  MoveL 760 to (-510.72, -291.87, 844) mm, rotated rx 180 ry 0 rz -90 deg; joints [21.183, -72.621, -92.099, -15.28, 68.817, -90]
  MoveL 761 to (-508.3, -277.31, 840) mm, rotated rx 180 ry 0 rz -90 deg; joints [21.364, -72.698, -94.24, -13.063, 68.636, -90]
  MoveL 762 to (-516.77, -268.54, 854) mm, rotated rx 180 ry 0 rz -90 deg; joints [20.699, -70.474, -96.997, -12.53, 69.301, -90]
  MoveL 763 to (-516.77, -255.15, 854) mm, rotated rx 180 ry 0 rz -90 deg; joints [20.699, -70.107, -99.223, -10.67, 69.301, -90]
  MoveL 764 to (-526.45, -246.29, 870) mm, rotated rx 180 ry 0 rz -90 deg; joints [19.827, -67.632, -102.031, -10.337, 70.173, -90]
  MoveL 765 to (-521.61, -230.51, 862) mm, rotated rx 180 ry 0 rz -90 deg; joints [20.28, -68.427, -103.896, -7.678, 69.72, -90]
  MoveL 766 to (-519.19, -215.98, 858) mm, rotated rx 180 ry 0 rz -90 deg; joints [20.493, -68.776, -105.82, -5.404, 69.507, -90]
  MoveL 767 to (-527.05, -205.6, 871) mm, rotated rx 180 ry 0 rz -90 deg; joints [19.768, -66.744, -108.538, -4.718, 70.232, -90]
  MoveL 768 to (-525.24, -191.28, 868) mm, rotated rx 180 ry 0 rz -90 deg; joints [19.944, -67.058, -110.452, -2.489, 70.056, -90]
  MoveL 769 to (-524.63, -177.46, 867) mm, rotated rx 180 ry 0 rz -90 deg; joints [20.001, -67.158, -112.413, -0.43, 69.999, -90]
  MoveL 770 to (-527.66, -164.81, 872) mm, rotated rx 180 ry 0 rz -90 deg; joints [19.709, -66.408, -114.69, 1.097, 70.291, -90]
  MoveL 771 to (-528.26, -151.31, 873) mm, rotated rx 180 ry 0 rz -90 deg; joints [19.649, -66.326, -116.708, 3.035, 70.351, -90]
  MoveL 772 to (-527.66, -137.46, 872) mm, rotated rx 180 ry 0 rz -90 deg; joints [19.709, -66.634, -118.561, 5.195, 70.291, -90]
  MoveL 773 to (-533.71, -125.21, 882) mm, rotated rx 180 ry 0 rz -90 deg; joints [19.079, -65.242, -121.134, 6.376, 70.921, -90]
  MoveL 774 to (-526.45, -109.86, 870) mm, rotated rx 180 ry 0 rz -90 deg; joints [19.827, -67.51, -122.122, 9.633, 70.173, -90]
  MoveL 775 to (-527.66, -96.44, 872) mm, rotated rx 180 ry 0 rz -90 deg; joints [19.709, -67.583, -124.075, 11.657, 70.291, -90]
  MoveL 776 to (-521.61, -81.82, 862) mm, rotated rx 180 ry 0 rz -90 deg; joints [20.28, -69.783, -124.958, 14.74, 69.72, -90]
  MoveL 777 to (-528.26, -69.17, 873) mm, rotated rx 180 ry 0 rz -90 deg; joints [19.649, -68.506, -127.639, 16.145, 70.351, -90]
  MoveL 778 to (-520.4, -54.65, 860) mm, rotated rx 180 ry 0 rz -90 deg; joints [20.388, -71.46, -128.062, 19.522, 69.612, -90]
  MoveL 779 to (-517.98, -40.98, 856) mm, rotated rx 180 ry 0 rz -90 deg; joints [20.597, -72.977, -129.219, 22.196, 69.403, -90]
  MoveL 780 to (-511.93, -27.23, 846) mm, rotated rx 180 ry 0 rz -90 deg; joints [21.089, -75.629, -129.608, 25.237, 68.911, -90]
  MoveL 781 to (-506.48, -13.82, 837) mm, rotated rx 180 ry 0 rz -90 deg; joints [21.496, -78.189, -129.943, 28.132, 68.504, -90]
  MoveL 782 to (-507.69, -0.69, 839) mm, rotated rx 180 ry 0 rz -90 deg; joints [21.409, -79.002, -131.528, 30.53, 68.591, -90]
  MoveL 783 to (-504.66, 12.39, 834) mm, rotated rx 180 ry 0 rz -90 deg; joints [21.625, -81.074, -132.163, 33.237, 68.375, -90]
  MoveL 784 to (-503.45, 25.41, 832) mm, rotated rx 180 ry 0 rz -90 deg; joints [21.709, -82.751, -133.104, 35.855, 68.291, -90]
  MoveL 785 to (-498.61, 38.08, 824) mm, rotated rx 180 ry 0 rz -90 deg; joints [22.032, -85.434, -133.121, 38.554, 67.969, -90]
  MoveL 786 to (-496.19, 50.76, 820) mm, rotated rx 180 ry 0 rz -90 deg; joints [22.185, -87.555, -133.593, 41.148, 67.815, -90]
  MoveL 787 to (-491.35, 63, 812) mm, rotated rx 180 ry 0 rz -90 deg; joints [22.478, -90.28, -133.363, 43.643, 67.522, -90]
  MoveL 788 to (-489.54, 75.45, 809) mm, rotated rx 180 ry 0 rz -90 deg; joints [22.583, -92.346, -133.791, 46.137, 67.418, -90]
  MoveL 789 to (-481.67, 86.72, 796) mm, rotated rx 180 ry 0 rz -90 deg; joints [23.011, -95.661, -132.528, 48.189, 66.989, -90]
  MoveL 790 to (-479.85, 98.83, 793) mm, rotated rx 180 ry 0 rz -90 deg; joints [23.104, -97.738, -132.762, 50.5, 66.896, -90]
  MoveL 791 to (-478.04, 110.84, 790) mm, rotated rx 180 ry 0 rz -90 deg; joints [23.195, -99.846, -132.917, 52.764, 66.805, -90]
  MoveL 792 to (-476.22, 122.76, 787) mm, rotated rx 180 ry 0 rz -90 deg; joints [23.284, -101.979, -132.995, 54.974, 66.717, -90]
  MoveL 793 to (-499.84, -492.72, 848) mm, rotated rx 180 ry 0 rz -90 deg; joints [23.844, -86.996, -46.335, -46.669, 66.156, -90]
  MoveL 794 to (-495.71, -475.46, 841) mm, rotated rx 180 ry 0 rz -90 deg; joints [24.056, -85.782, -50.992, -43.226, 65.944, -90]
  MoveL 795 to (-492.18, -458.98, 835) mm, rotated rx 180 ry 0 rz -90 deg; joints [24.228, -84.764, -55.111, -40.125, 65.772, -90]
  MoveL 796 to (-498.07, -451.22, 845) mm, rotated rx 180 ry 0 rz -90 deg; joints [23.937, -82.603, -58.407, -38.99, 66.063, -90]
  MoveL 797 to (-496.89, -436.94, 843) mm, rotated rx 180 ry 0 rz -90 deg; joints [23.997, -81.512, -61.93, -36.557, 66.003, -90]
  MoveL 798 to (-491.59, -419.19, 834) mm, rotated rx 180 ry 0 rz -90 deg; joints [24.256, -81.2, -65.344, -33.456, 65.744, -90]
  MoveL 799 to (-494.53, -408.55, 839) mm, rotated rx 180 ry 0 rz -90 deg; joints [24.114, -79.678, -68.387, -31.935, 65.886, -90]
  MoveL 800 to (-490.41, -392.09, 832) mm, rotated rx 180 ry 0 rz -90 deg; joints [24.311, -79.429, -71.37, -29.201, 65.69, -90]
  MoveL 801 to (-491, -379.5, 833) mm, rotated rx 180 ry 0 rz -90 deg; joints [24.283, -78.45, -74.205, -27.345, 65.717, -90]
  MoveL 802 to (-492.18, -367.32, 835) mm, rotated rx 180 ry 0 rz -90 deg; joints [24.228, -77.42, -76.962, -25.618, 65.772, -90]
  MoveL 803 to (-491.59, -353.8, 834) mm, rotated rx 180 ry 0 rz -90 deg; joints [24.256, -76.782, -79.601, -23.616, 65.744, -90]
  MoveL 804 to (-494.53, -342.77, 839) mm, rotated rx 180 ry 0 rz -90 deg; joints [24.114, -75.504, -82.269, -22.227, 65.886, -90]
  MoveL 805 to (-492.76, -328.43, 836) mm, rotated rx 180 ry 0 rz -90 deg; joints [24.2, -75.22, -84.714, -20.066, 65.8, -90]
  MoveL 806 to (-498.66, -319.09, 846) mm, rotated rx 180 ry 0 rz -90 deg; joints [23.906, -73.399, -87.416, -19.185, 66.094, -90]
  MoveL 807 to (-497.48, -305.1, 844) mm, rotated rx 180 ry 0 rz -90 deg; joints [23.967, -73.091, -89.772, -17.136, 66.033, -90]
  MoveL 808 to (-499.84, -293.25, 848) mm, rotated rx 180 ry 0 rz -90 deg; joints [23.844, -72.074, -92.25, -15.676, 66.156, -90]
  MoveL 809 to (-496.89, -278.3, 843) mm, rotated rx 180 ry 0 rz -90 deg; joints [23.997, -72.283, -94.367, -13.35, 66.003, -90]
  MoveL 810 to (-497.48, -265.4, 844) mm, rotated rx 180 ry 0 rz -90 deg; joints [23.967, -71.761, -96.64, -11.599, 66.033, -90]
  MoveL 811 to (-506.32, -256.64, 859) mm, rotated rx 180 ry 0 rz -90 deg; joints [23.482, -69.341, -99.474, -11.185, 66.518, -90]
  MoveL 812 to (-511.63, -245.72, 868) mm, rotated rx 180 ry 0 rz -90 deg; joints [23.156, -67.749, -102.047, -10.204, 66.844, -90]
  MoveL 813 to (-510.45, -231.58, 866) mm, rotated rx 180 ry 0 rz -90 deg; joints [23.231, -67.732, -104.149, -8.119, 66.769, -90]
  MoveL 814 to (-513.98, -219.51, 872) mm, rotated rx 180 ry 0 rz -90 deg; joints [23.002, -66.616, -106.57, -6.815, 66.998, -90]
  MoveL 815 to (-513.98, -205.83, 872) mm, rotated rx 180 ry 0 rz -90 deg; joints [23.002, -66.418, -108.688, -4.893, 66.998, -90]
  MoveL 816 to (-509.27, -190.39, 864) mm, rotated rx 180 ry 0 rz -90 deg; joints [23.304, -67.515, -110.316, -2.169, 66.696, -90]
  MoveL 817 to (-512.81, -178.07, 870) mm, rotated rx 180 ry 0 rz -90 deg; joints [23.08, -66.53, -112.683, -0.786, 66.92, -90]
  MoveL 818 to (-512.81, -164.43, 870) mm, rotated rx 180 ry 0 rz -90 deg; joints [23.08, -66.538, -114.671, 1.209, 66.92, -90]
  MoveL 819 to (-510.45, -150.1, 866) mm, rotated rx 180 ry 0 rz -90 deg; joints [23.231, -67.272, -116.344, 3.616, 66.769, -90]
  MoveL 820 to (-515.75, -137.93, 875) mm, rotated rx 180 ry 0 rz -90 deg; joints [22.882, -65.937, -118.884, 4.821, 67.118, -90]
  MoveL 821 to (-516.34, -124.35, 876) mm, rotated rx 180 ry 0 rz -90 deg; joints [22.841, -65.986, -120.85, 6.836, 67.159, -90]
  MoveL 822 to (-519.29, -111.25, 881) mm, rotated rx 180 ry 0 rz -90 deg; joints [22.631, -65.421, -123.091, 8.512, 67.369, -90]
  MoveL 823 to (-513.98, -96.44, 872) mm, rotated rx 180 ry 0 rz -90 deg; joints [23.002, -67.378, -124.193, 11.57, 66.998, -90]
  MoveL 824 to (-510.45, -82.2, 866) mm, rotated rx 180 ry 0 rz -90 deg; joints [23.231, -68.937, -125.412, 14.35, 66.769, -90]
  MoveL 825 to (-512.22, -68.85, 869) mm, rotated rx 180 ry 0 rz -90 deg; joints [23.118, -69.007, -127.391, 16.398, 66.882, -90]
  MoveL 826 to (-509.27, -54.91, 864) mm, rotated rx 180 ry 0 rz -90 deg; joints [23.304, -70.615, -128.553, 19.168, 66.696, -90]
  MoveL 827 to (-503.37, -40.88, 854) mm, rotated rx 180 ry 0 rz -90 deg; joints [23.651, -73.232, -129.066, 22.298, 66.349, -90]
  MoveL 828 to (-498.07, -27.2, 845) mm, rotated rx 180 ry 0 rz -90 deg; joints [23.937, -75.76, -129.521, 25.281, 66.063, -90]
  MoveL 829 to (-495.12, -13.87, 840) mm, rotated rx 180 ry 0 rz -90 deg; joints [24.086, -77.673, -130.319, 27.992, 65.914, -90]
  MoveL 830 to (-491.59, -0.69, 834) mm, rotated rx 180 ry 0 rz -90 deg; joints [24.256, -79.841, -130.884, 30.725, 65.744, -90]
  MoveL 831 to (-492.76, 12.42, 836) mm, rotated rx 180 ry 0 rz -90 deg; joints [24.2, -80.756, -132.421, 33.177, 65.8, -90]
  MoveL 832 to (-491.59, 25.47, 834) mm, rotated rx 180 ry 0 rz -90 deg; joints [24.256, -82.45, -133.364, 35.814, 65.744, -90]
  MoveL 833 to (-484.51, 37.99, 822) mm, rotated rx 180 ry 0 rz -90 deg; joints [24.571, -85.795, -132.78, 38.575, 65.429, -90]
  MoveL 834 to (-479.8, 50.39, 814) mm, rotated rx 180 ry 0 rz -90 deg; joints [24.765, -88.502, -132.621, 41.123, 65.235, -90]
  MoveL 835 to (-478.62, 63, 812) mm, rotated rx 180 ry 0 rz -90 deg; joints [24.811, -90.369, -133.273, 43.642, 65.189, -90]
  MoveL 836 to (-476.26, 75.36, 808) mm, rotated rx 180 ry 0 rz -90 deg; joints [24.902, -92.572, -133.53, 46.102, 65.098, -90]
  MoveL 837 to (-468.6, 86.61, 795) mm, rotated rx 180 ry 0 rz -90 deg; joints [25.178, -95.905, -132.221, 48.125, 64.822, -90]
  MoveL 838 to (-466.83, 98.7, 792) mm, rotated rx 180 ry 0 rz -90 deg; joints [25.239, -97.975, -132.441, 50.416, 64.761, -90]
  MoveL 839 to (-466.83, 111.12, 792) mm, rotated rx 180 ry 0 rz -90 deg; joints [25.239, -99.763, -133.094, 52.857, 64.761, -90]
  MoveL 840 to (-468.01, 123.86, 794) mm, rotated rx 180 ry 0 rz -90 deg; joints [25.199, -101.44, -134.021, 55.461, 64.801, -90]
  MoveL 841 to (-483.67, -489.81, 843) mm, rotated rx 180 ry 0 rz -90 deg; joints [26.705, -87.373, -46.601, -46.025, 63.295, -90]
  MoveL 842 to (-485.39, -478.29, 846) mm, rotated rx 180 ry 0 rz -90 deg; joints [26.662, -85.483, -50.688, -43.829, 63.338, -90]
  MoveL 843 to (-483.67, -463.37, 843) mm, rotated rx 180 ry 0 rz -90 deg; joints [26.705, -84.199, -54.753, -41.047, 63.295, -90]
  MoveL 844 to (-480.8, -447.49, 838) mm, rotated rx 180 ry 0 rz -90 deg; joints [26.775, -83.263, -58.557, -38.179, 63.225, -90]
  MoveL 845 to (-483.1, -436.42, 842) mm, rotated rx 180 ry 0 rz -90 deg; joints [26.72, -81.666, -61.901, -36.433, 63.28, -90]
  MoveL 846 to (-481.95, -422.21, 840) mm, rotated rx 180 ry 0 rz -90 deg; joints [26.748, -80.707, -65.206, -34.087, 63.252, -90]
  MoveL 847 to (-480.23, -407.58, 837) mm, rotated rx 180 ry 0 rz -90 deg; joints [26.789, -79.957, -68.338, -31.705, 63.211, -90]
  MoveL 848 to (-477.36, -392.09, 832) mm, rotated rx 180 ry 0 rz -90 deg; joints [26.855, -79.528, -71.294, -29.179, 63.145, -90]
  MoveL 849 to (-478.51, -379.96, 834) mm, rotated rx 180 ry 0 rz -90 deg; joints [26.829, -78.435, -74.142, -27.423, 63.171, -90]
  MoveL 850 to (-478.51, -366.88, 834) mm, rotated rx 180 ry 0 rz -90 deg; joints [26.829, -77.624, -76.882, -25.494, 63.171, -90]
  MoveL 851 to (-482.52, -356.77, 841) mm, rotated rx 180 ry 0 rz -90 deg; joints [26.734, -76.054, -79.653, -24.293, 63.266, -90]
  MoveL 852 to (-480.8, -342.36, 838) mm, rotated rx 180 ry 0 rz -90 deg; joints [26.775, -75.702, -82.193, -22.105, 63.225, -90]
  MoveL 853 to (-484.25, -331.57, 844) mm, rotated rx 180 ry 0 rz -90 deg; joints [26.691, -74.315, -84.854, -20.831, 63.309, -90]
  MoveL 854 to (-483.67, -317.96, 843) mm, rotated rx 180 ry 0 rz -90 deg; joints [26.705, -73.833, -87.297, -18.87, 63.295, -90]
  MoveL 855 to (-485.97, -306.19, 847) mm, rotated rx 180 ry 0 rz -90 deg; joints [26.647, -72.763, -89.826, -17.411, 63.353, -90]
  MoveL 856 to (-486.54, -293.25, 848) mm, rotated rx 180 ry 0 rz -90 deg; joints [26.632, -72.121, -92.219, -15.66, 63.368, -90]
  MoveL 857 to (-485.39, -279.29, 846) mm, rotated rx 180 ry 0 rz -90 deg; joints [26.662, -71.938, -94.445, -13.617, 63.338, -90]
  MoveL 858 to (-484.25, -265.4, 844) mm, rotated rx 180 ry 0 rz -90 deg; joints [26.691, -71.825, -96.598, -11.577, 63.309, -90]
  MoveL 859 to (-490.56, -255.45, 855) mm, rotated rx 180 ry 0 rz -90 deg; joints [26.524, -69.914, -99.299, -10.788, 63.476, -90]
  MoveL 860 to (-494, -243.74, 861) mm, rotated rx 180 ry 0 rz -90 deg; joints [26.425, -68.724, -101.763, -9.513, 63.575, -90]
  MoveL 861 to (-499.74, -232.91, 871) mm, rotated rx 180 ry 0 rz -90 deg; joints [26.247, -66.961, -104.398, -8.641, 63.753, -90]
  MoveL 862 to (-502.03, -220.26, 875) mm, rotated rx 180 ry 0 rz -90 deg; joints [26.171, -66.1, -106.749, -7.152, 63.829, -90]
  MoveL 863 to (-505.47, -207.96, 881) mm, rotated rx 180 ry 0 rz -90 deg; joints [26.05, -64.963, -109.181, -5.857, 63.95, -90]
  MoveL 864 to (-500.88, -192.38, 873) mm, rotated rx 180 ry 0 rz -90 deg; joints [26.21, -66.062, -110.858, -3.08, 63.791, -90]
  MoveL 865 to (-500.31, -178.48, 872) mm, rotated rx 180 ry 0 rz -90 deg; joints [26.229, -66.152, -112.838, -1.011, 63.771, -90]
  MoveL 866 to (-496.87, -163.68, 866) mm, rotated rx 180 ry 0 rz -90 deg; joints [26.339, -67.148, -114.431, 1.579, 63.661, -90]
  MoveL 867 to (-502.03, -151.66, 875) mm, rotated rx 180 ry 0 rz -90 deg; joints [26.171, -65.714, -117, 2.714, 63.829, -90]
  MoveL 868 to (-500.31, -137.46, 872) mm, rotated rx 180 ry 0 rz -90 deg; joints [26.229, -66.37, -118.711, 5.081, 63.771, -90]
  MoveL 869 to (-500.88, -123.93, 873) mm, rotated rx 180 ry 0 rz -90 deg; joints [26.21, -66.42, -120.669, 7.09, 63.791, -90]
  MoveL 870 to (-509.49, -112.13, 888) mm, rotated rx 180 ry 0 rz -90 deg; joints [25.899, -64.03, -123.702, 7.732, 64.101, -90]
  MoveL 871 to (-502.03, -96.77, 875) mm, rotated rx 180 ry 0 rz -90 deg; joints [26.171, -66.761, -124.495, 11.256, 63.829, -90]
  MoveL 872 to (-499.74, -82.67, 871) mm, rotated rx 180 ry 0 rz -90 deg; joints [26.247, -67.985, -125.903, 13.888, 63.753, -90]
  MoveL 873 to (-504.9, -69.72, 880) mm, rotated rx 180 ry 0 rz -90 deg; joints [26.071, -66.898, -128.476, 15.374, 63.929, -90]
  MoveL 874 to (-493.43, -54.65, 860) mm, rotated rx 180 ry 0 rz -90 deg; joints [26.442, -71.331, -128.144, 19.475, 63.558, -90]
  MoveL 875 to (-492.85, -41.12, 859) mm, rotated rx 180 ry 0 rz -90 deg; joints [26.459, -72.341, -129.611, 21.952, 63.541, -90]
  MoveL 876 to (-488.26, -27.39, 851) mm, rotated rx 180 ry 0 rz -90 deg; joints [26.587, -74.747, -130.195, 24.942, 63.413, -90]
  MoveL 877 to (-481.38, -13.85, 839) mm, rotated rx 180 ry 0 rz -90 deg; joints [26.762, -77.941, -130.123, 28.064, 63.238, -90]
  MoveL 878 to (-483.1, -0.7, 842) mm, rotated rx 180 ry 0 rz -90 deg; joints [26.72, -78.563, -131.859, 30.422, 63.28, -90]
  MoveL 879 to (-481.38, 12.46, 839) mm, rotated rx 180 ry 0 rz -90 deg; joints [26.762, -80.349, -132.75, 33.098, 63.238, -90]
  MoveL 880 to (-475.64, 25.32, 829) mm, rotated rx 180 ry 0 rz -90 deg; joints [26.894, -83.385, -132.556, 35.941, 63.106, -90]
  MoveL 881 to (-471.62, 37.99, 822) mm, rotated rx 180 ry 0 rz -90 deg; joints [26.98, -85.942, -132.648, 38.59, 63.02, -90]
  MoveL 882 to (-469.9, 50.7, 819) mm, rotated rx 180 ry 0 rz -90 deg; joints [27.015, -87.921, -133.236, 41.157, 62.985, -90]
  MoveL 883 to (-464.74, 62.84, 810) mm, rotated rx 180 ry 0 rz -90 deg; joints [27.116, -90.816, -132.788, 43.604, 62.884, -90]
  MoveL 884 to (-468.18, 76.1, 816) mm, rotated rx 180 ry 0 rz -90 deg; joints [27.05, -91.668, -134.644, 46.312, 62.95, -90]
  MoveL 885 to (-459.57, 87.26, 801) mm, rotated rx 180 ry 0 rz -90 deg; joints [27.21, -95.351, -133.005, 48.357, 62.79, -90]
  MoveL 886 to (-455.56, 98.95, 794) mm, rotated rx 180 ry 0 rz -90 deg; joints [27.279, -97.93, -132.554, 50.484, 62.721, -90]
  MoveL 887 to (-452.12, 110.56, 788) mm, rotated rx 180 ry 0 rz -90 deg; joints [27.336, -100.36, -132.175, 52.535, 62.664, -90]
  MoveL 888 to (-454.98, 123.7, 793) mm, rotated rx 180 ry 0 rz -90 deg; joints [27.289, -101.7, -133.621, 55.321, 62.711, -90]
  MoveL 889 to (-470.45, -489.81, 843) mm, rotated rx 180 ry 0 rz -90 deg; joints [29.342, -87.528, -46.458, -46.015, 60.658, -90]
  MoveL 890 to (-472.13, -478.29, 846) mm, rotated rx 180 ry 0 rz -90 deg; joints [29.344, -85.625, -50.563, -43.812, 60.656, -90]
  MoveL 891 to (-474.36, -467.22, 850) mm, rotated rx 180 ry 0 rz -90 deg; joints [29.348, -83.774, -54.365, -41.861, 60.652, -90]
  MoveL 892 to (-472.13, -451.76, 846) mm, rotated rx 180 ry 0 rz -90 deg; joints [29.344, -82.713, -58.216, -39.071, 60.656, -90]
  MoveL 893 to (-469.89, -436.42, 842) mm, rotated rx 180 ry 0 rz -90 deg; joints [29.341, -81.816, -61.78, -36.404, 60.659, -90]
  MoveL 894 to (-468.22, -421.71, 839) mm, rotated rx 180 ry 0 rz -90 deg; joints [29.339, -80.962, -65.093, -33.945, 60.661, -90]
  MoveL 895 to (-471.01, -410.98, 844) mm, rotated rx 180 ry 0 rz -90 deg; joints [29.343, -79.396, -68.184, -32.421, 60.657, -90]
  MoveL 896 to (-463.2, -391.15, 830) mm, rotated rx 180 ry 0 rz -90 deg; joints [29.332, -79.926, -71.141, -28.933, 60.668, -90]
  MoveL 897 to (-469.89, -383.6, 842) mm, rotated rx 180 ry 0 rz -90 deg; joints [29.341, -77.709, -74.083, -28.209, 60.659, -90]
  MoveL 898 to (-471.01, -371.28, 844) mm, rotated rx 180 ry 0 rz -90 deg; joints [29.343, -76.637, -76.89, -26.473, 60.657, -90]
  MoveL 899 to (-471.01, -358.04, 844) mm, rotated rx 180 ry 0 rz -90 deg; joints [29.343, -75.852, -79.592, -24.556, 60.657, -90]
  MoveL 900 to (-465.43, -340.72, 834) mm, rotated rx 180 ry 0 rz -90 deg; joints [29.335, -76.364, -81.975, -21.661, 60.665, -90]
  MoveL 901 to (-472.13, -332.36, 846) mm, rotated rx 180 ry 0 rz -90 deg; joints [29.344, -74.211, -84.803, -20.986, 60.656, -90]
  MoveL 902 to (-471.01, -318.34, 844) mm, rotated rx 180 ry 0 rz -90 deg; joints [29.343, -73.856, -87.223, -18.921, 60.657, -90]
  MoveL 903 to (-477.15, -309.08, 855) mm, rotated rx 180 ry 0 rz -90 deg; joints [29.352, -71.846, -89.982, -18.172, 60.648, -90]
  MoveL 904 to (-478.82, -296.71, 858) mm, rotated rx 180 ry 0 rz -90 deg; joints [29.355, -70.904, -92.475, -16.621, 60.645, -90]
  MoveL 905 to (-473.24, -279.95, 848) mm, rotated rx 180 ry 0 rz -90 deg; joints [29.346, -71.806, -94.432, -13.762, 60.654, -90]
  MoveL 906 to (-479.94, -270.43, 860) mm, rotated rx 180 ry 0 rz -90 deg; joints [29.357, -69.692, -97.2, -13.108, 60.643, -90]
  MoveL 907 to (-478.27, -256.05, 857) mm, rotated rx 180 ry 0 rz -90 deg; joints [29.354, -69.742, -99.316, -10.942, 60.646, -90]
  MoveL 908 to (-486.64, -246.85, 872) mm, rotated rx 180 ry 0 rz -90 deg; joints [29.369, -67.187, -102.204, -10.609, 60.631, -90]
  MoveL 909 to (-488.31, -233.98, 875) mm, rotated rx 180 ry 0 rz -90 deg; joints [29.372, -66.413, -104.55, -9.037, 60.628, -90]
  MoveL 910 to (-488.87, -220.51, 876) mm, rotated rx 180 ry 0 rz -90 deg; joints [29.373, -65.987, -106.775, -7.239, 60.627, -90]
  MoveL 911 to (-488.31, -206.54, 875) mm, rotated rx 180 ry 0 rz -90 deg; joints [29.372, -65.934, -108.856, -5.21, 60.628, -90]
  MoveL 912 to (-488.31, -192.82, 875) mm, rotated rx 180 ry 0 rz -90 deg; joints [29.372, -65.788, -110.946, -3.266, 60.628, -90]
  MoveL 913 to (-487.75, -178.89, 874) mm, rotated rx 180 ry 0 rz -90 deg; joints [29.371, -65.876, -112.932, -1.192, 60.629, -90]
  MoveL 914 to (-485.52, -164.43, 870) mm, rotated rx 180 ry 0 rz -90 deg; joints [29.367, -66.553, -114.663, 1.215, 60.634, -90]
  MoveL 915 to (-491.66, -152.7, 881) mm, rotated rx 180 ry 0 rz -90 deg; joints [29.379, -64.711, -117.395, 2.106, 60.621, -90]
  MoveL 916 to (-487.75, -137.78, 874) mm, rotated rx 180 ry 0 rz -90 deg; joints [29.371, -66.076, -118.83, 4.905, 60.629, -90]
  MoveL 917 to (-489.98, -124.64, 878) mm, rotated rx 180 ry 0 rz -90 deg; joints [29.375, -65.571, -121.038, 6.608, 60.625, -90]
  MoveL 918 to (-492.77, -111.5, 883) mm, rotated rx 180 ry 0 rz -90 deg; joints [29.381, -64.935, -123.317, 8.252, 60.619, -90]
  MoveL 919 to (-489.98, -97.1, 878) mm, rotated rx 180 ry 0 rz -90 deg; joints [29.375, -66.246, -124.733, 10.98, 60.625, -90]
  MoveL 920 to (-486.64, -82.76, 872) mm, rotated rx 180 ry 0 rz -90 deg; joints [29.369, -67.867, -125.957, 13.824, 60.631, -90]
  MoveL 921 to (-482.73, -68.54, 865) mm, rotated rx 180 ry 0 rz -90 deg; joints [29.362, -69.794, -126.965, 16.759, 60.638, -90]
  MoveL 922 to (-477.15, -54.34, 855) mm, rotated rx 180 ry 0 rz -90 deg; joints [29.352, -72.394, -127.511, 19.905, 60.648, -90]
  MoveL 923 to (-478.82, -41.07, 858) mm, rotated rx 180 ry 0 rz -90 deg; joints [29.355, -72.659, -129.412, 22.071, 60.645, -90]
  MoveL 924 to (-474.92, -27.39, 851) mm, rotated rx 180 ry 0 rz -90 deg; joints [29.349, -74.907, -130.084, 24.992, 60.651, -90]
  MoveL 925 to (-472.13, -13.96, 846) mm, rotated rx 180 ry 0 rz -90 deg; joints [29.344, -76.875, -130.885, 27.76, 60.656, -90]
  MoveL 926 to (-472.13, -0.7, 846) mm, rotated rx 180 ry 0 rz -90 deg; joints [29.344, -78.035, -132.252, 30.287, 60.656, -90]
  MoveL 927 to (-465.43, 12.39, 834) mm, rotated rx 180 ry 0 rz -90 deg; joints [29.335, -81.412, -131.892, 33.304, 60.665, -90]
  MoveL 928 to (-458.73, 25.1, 822) mm, rotated rx 180 ry 0 rz -90 deg; joints [29.327, -84.757, -131.335, 36.092, 60.673, -90]
  MoveL 929 to (-456.5, 37.81, 818) mm, rotated rx 180 ry 0 rz -90 deg; joints [29.324, -86.804, -131.827, 38.631, 60.676, -90]
  MoveL 930 to (-457.06, 50.7, 819) mm, rotated rx 180 ry 0 rz -90 deg; joints [29.325, -88.153, -133.015, 41.168, 60.675, -90]
  MoveL 931 to (-454.27, 63.15, 814) mm, rotated rx 180 ry 0 rz -90 deg; joints [29.321, -90.486, -133.187, 43.672, 60.679, -90]
  MoveL 932 to (-452.59, 75.64, 811) mm, rotated rx 180 ry 0 rz -90 deg; joints [29.32, -92.573, -133.588, 46.161, 60.68, -90]
  MoveL 933 to (-447.57, 87.37, 802) mm, rotated rx 180 ry 0 rz -90 deg; joints [29.314, -95.464, -132.899, 48.363, 60.686, -90]
  MoveL 934 to (-442.55, 98.83, 793) mm, rotated rx 180 ry 0 rz -90 deg; joints [29.309, -98.282, -132.088, 50.371, 60.691, -90]
  MoveL 935 to (-440.32, 110.7, 789) mm, rotated rx 180 ry 0 rz -90 deg; joints [29.307, -100.488, -132.04, 52.528, 60.693, -90]
  MoveL 936 to (-441.99, 123.54, 792) mm, rotated rx 180 ry 0 rz -90 deg; joints [29.309, -102.015, -133.144, 55.159, 60.691, -90]
  MoveL 937 to (-459.94, -492.72, 848) mm, rotated rx 180 ry 0 rz -90 deg; joints [31.975, -87.41, -45.953, -46.637, 58.025, -90]
  MoveL 938 to (-460.49, -479.99, 849) mm, rotated rx 180 ry 0 rz -90 deg; joints [31.991, -85.62, -50.223, -44.157, 58.009, -90]
  MoveL 939 to (-462.66, -468.87, 853) mm, rotated rx 180 ry 0 rz -90 deg; joints [32.056, -83.74, -54.069, -42.191, 57.944, -90]
  MoveL 940 to (-456.15, -449.09, 841) mm, rotated rx 180 ry 0 rz -90 deg; joints [31.867, -83.393, -58.151, -38.457, 58.133, -90]
  MoveL 941 to (-456.15, -435.9, 841) mm, rotated rx 180 ry 0 rz -90 deg; joints [31.867, -82.146, -61.606, -36.248, 58.133, -90]
  MoveL 942 to (-456.15, -422.71, 841) mm, rotated rx 180 ry 0 rz -90 deg; joints [31.867, -80.998, -64.887, -34.115, 58.133, -90]
  MoveL 943 to (-457.78, -410.98, 844) mm, rotated rx 180 ry 0 rz -90 deg; joints [31.912, -79.623, -68.009, -32.367, 58.088, -90]
  MoveL 944 to (-456.15, -396.33, 841) mm, rotated rx 180 ry 0 rz -90 deg; joints [31.867, -78.961, -71.016, -30.023, 58.133, -90]
  MoveL 945 to (-459.94, -386.34, 848) mm, rotated rx 180 ry 0 rz -90 deg; joints [31.975, -77.263, -73.955, -28.782, 58.025, -90]
  MoveL 946 to (-455.61, -369.52, 840) mm, rotated rx 180 ry 0 rz -90 deg; joints [31.852, -77.338, -76.666, -25.996, 58.148, -90]
  MoveL 947 to (-456.69, -357.2, 842) mm, rotated rx 180 ry 0 rz -90 deg; joints [31.882, -76.326, -79.39, -24.284, 58.118, -90]
  MoveL 948 to (-454.52, -342.36, 838) mm, rotated rx 180 ry 0 rz -90 deg; joints [31.823, -76.114, -81.898, -21.988, 58.177, -90]
  MoveL 949 to (-458.86, -332.36, 846) mm, rotated rx 180 ry 0 rz -90 deg; joints [31.943, -74.441, -84.645, -20.914, 58.057, -90]
  MoveL 950 to (-461.57, -320.98, 851) mm, rotated rx 180 ry 0 rz -90 deg; joints [32.023, -73.17, -87.278, -19.552, 57.977, -90]
  MoveL 951 to (-467, -311.25, 861) mm, rotated rx 180 ry 0 rz -90 deg; joints [32.195, -71.252, -90.028, -18.72, 57.805, -90]
  MoveL 952 to (-465.37, -296.71, 858) mm, rotated rx 180 ry 0 rz -90 deg; joints [32.141, -71.108, -92.346, -16.545, 57.859, -90]
  MoveL 953 to (-461.03, -280.61, 850) mm, rotated rx 180 ry 0 rz -90 deg; joints [32.007, -71.755, -94.366, -13.879, 57.993, -90]
  MoveL 954 to (-469.71, -272.32, 866) mm, rotated rx 180 ry 0 rz -90 deg; joints [32.287, -69.026, -97.321, -13.652, 57.713, -90]
  MoveL 955 to (-471.88, -259.93, 870) mm, rotated rx 180 ry 0 rz -90 deg; joints [32.364, -68.026, -99.77, -12.204, 57.636, -90]
  MoveL 956 to (-472.96, -246.85, 872) mm, rotated rx 180 ry 0 rz -90 deg; joints [32.404, -67.356, -102.107, -10.538, 57.596, -90]
  MoveL 957 to (-474.59, -233.98, 875) mm, rotated rx 180 ry 0 rz -90 deg; joints [32.465, -66.573, -104.46, -8.967, 57.535, -90]
  MoveL 958 to (-477.84, -221.77, 881) mm, rotated rx 180 ry 0 rz -90 deg; joints [32.594, -65.348, -106.941, -7.712, 57.406, -90]
  MoveL 959 to (-485.44, -211.26, 895) mm, rotated rx 180 ry 0 rz -90 deg; joints [32.929, -62.825, -109.807, -7.368, 57.071, -90]
  MoveL 960 to (-478.93, -194.58, 883) mm, rotated rx 180 ry 0 rz -90 deg; joints [32.638, -64.616, -111.327, -4.057, 57.362, -90]
  MoveL 961 to (-477.84, -180.33, 881) mm, rotated rx 180 ry 0 rz -90 deg; joints [32.594, -64.851, -113.285, -1.864, 57.406, -90]
  MoveL 962 to (-475.67, -165.75, 877) mm, rotated rx 180 ry 0 rz -90 deg; joints [32.507, -65.522, -115.047, 0.569, 57.493, -90]
  MoveL 963 to (-481.64, -153.91, 888) mm, rotated rx 180 ry 0 rz -90 deg; joints [32.754, -63.603, -117.803, 1.406, 57.246, -90]
  MoveL 964 to (-482.72, -140.3, 890) mm, rotated rx 180 ry 0 rz -90 deg; joints [32.803, -63.325, -119.935, 3.26, 57.197, -90]
  MoveL 965 to (-477.84, -125.06, 881) mm, rotated rx 180 ry 0 rz -90 deg; joints [32.594, -65.181, -121.188, 6.368, 57.406, -90]
  MoveL 966 to (-476.76, -111, 879) mm, rotated rx 180 ry 0 rz -90 deg; joints [32.55, -65.846, -122.896, 8.742, 57.45, -90]
  MoveL 967 to (-474.59, -96.77, 875) mm, rotated rx 180 ry 0 rz -90 deg; joints [32.465, -66.997, -124.361, 11.358, 57.535, -90]
  MoveL 968 to (-476.22, -83.33, 878) mm, rotated rx 180 ry 0 rz -90 deg; joints [32.528, -66.903, -126.423, 13.325, 57.472, -90]
  MoveL 969 to (-471.33, -68.85, 869) mm, rotated rx 180 ry 0 rz -90 deg; joints [32.344, -69.25, -127.246, 16.496, 57.656, -90]
  MoveL 970 to (-461.57, -54.08, 851) mm, rotated rx 180 ry 0 rz -90 deg; joints [32.023, -73.412, -126.877, 20.289, 57.977, -90]
  MoveL 971 to (-460.49, -40.64, 849) mm, rotated rx 180 ry 0 rz -90 deg; joints [31.991, -74.619, -128.167, 22.786, 58.009, -90]
  MoveL 972 to (-462.66, -27.46, 853) mm, rotated rx 180 ry 0 rz -90 deg; joints [32.056, -74.805, -130.144, 24.949, 57.944, -90]
  MoveL 973 to (-461.03, -14.03, 850) mm, rotated rx 180 ry 0 rz -90 deg; joints [32.007, -76.42, -131.201, 27.621, 57.993, -90]
  MoveL 974 to (-459.4, -0.7, 847) mm, rotated rx 180 ry 0 rz -90 deg; joints [31.959, -78.138, -132.176, 30.314, 58.041, -90]
  MoveL 975 to (-457.78, 12.54, 844) mm, rotated rx 180 ry 0 rz -90 deg; joints [31.912, -79.956, -133.068, 33.025, 58.088, -90]
  MoveL 976 to (-447.47, 25.19, 825) mm, rotated rx 180 ry 0 rz -90 deg; joints [31.644, -84.581, -131.505, 36.086, 58.356, -90]
  MoveL 977 to (-448.01, 38.18, 826) mm, rotated rx 180 ry 0 rz -90 deg; joints [31.657, -85.845, -132.77, 38.615, 58.343, -90]
  MoveL 978 to (-445.84, 50.88, 822) mm, rotated rx 180 ry 0 rz -90 deg; joints [31.605, -88.003, -133.193, 41.197, 58.395, -90]
  MoveL 979 to (-440.42, 63, 812) mm, rotated rx 180 ry 0 rz -90 deg; joints [31.484, -91.081, -132.548, 43.629, 58.517, -90]
  MoveL 980 to (-438.79, 75.45, 809) mm, rotated rx 180 ry 0 rz -90 deg; joints [31.449, -93.146, -132.932, 46.077, 58.551, -90]
  MoveL 981 to (-433.91, 87.16, 800) mm, rotated rx 180 ry 0 rz -90 deg; joints [31.349, -96.014, -132.213, 48.226, 58.651, -90]
  MoveL 982 to (-433.91, 99.7, 800) mm, rotated rx 180 ry 0 rz -90 deg; joints [31.349, -97.759, -132.937, 50.695, 58.651, -90]
  MoveL 983 to (-428.49, 110.84, 790) mm, rotated rx 180 ry 0 rz -90 deg; joints [31.246, -100.663, -131.84, 52.504, 58.754, -90]
  MoveL 984 to (-431.2, 124.01, 795) mm, rotated rx 180 ry 0 rz -90 deg; joints [31.297, -101.988, -133.301, 55.289, 58.703, -90]
  MoveL 985 to (-448.23, -494.46, 851) mm, rotated rx 180 ry 0 rz -90 deg; joints [34.6, -87.512, -45.487, -47.002, 55.4, -90]
  MoveL 986 to (-450.33, -483.38, 855) mm, rotated rx 180 ry 0 rz -90 deg; joints [34.726, -85.457, -49.672, -44.871, 55.274, -90]
  MoveL 987 to (-446.65, -466.12, 848) mm, rotated rx 180 ry 0 rz -90 deg; joints [34.509, -84.464, -53.992, -41.544, 55.491, -90]
  MoveL 988 to (-445.07, -451.22, 845) mm, rotated rx 180 ry 0 rz -90 deg; joints [34.42, -83.338, -57.797, -38.865, 55.58, -90]
  MoveL 989 to (-436.11, -429.16, 828) mm, rotated rx 180 ry 0 rz -90 deg; joints [33.958, -83.771, -61.455, -34.775, 56.042, -90]
  MoveL 990 to (-444.01, -423.72, 843) mm, rotated rx 180 ry 0 rz -90 deg; joints [34.362, -81.108, -64.622, -34.27, 55.638, -90]
  MoveL 991 to (-444.54, -410.98, 844) mm, rotated rx 180 ry 0 rz -90 deg; joints [34.391, -79.933, -67.77, -32.297, 55.609, -90]
  MoveL 992 to (-445.59, -398.69, 846) mm, rotated rx 180 ry 0 rz -90 deg; joints [34.449, -78.721, -70.8, -30.479, 55.551, -90]
  MoveL 993 to (-446.65, -386.34, 848) mm, rotated rx 180 ry 0 rz -90 deg; joints [34.509, -77.567, -73.733, -28.7, 55.491, -90]
  MoveL 994 to (-442.43, -369.52, 840) mm, rotated rx 180 ry 0 rz -90 deg; joints [34.277, -77.659, -76.429, -25.912, 55.723, -90]
  MoveL 995 to (-445.07, -358.47, 845) mm, rotated rx 180 ry 0 rz -90 deg; joints [34.42, -76.275, -79.222, -24.503, 55.58, -90]
  MoveL 996 to (-444.01, -344.4, 843) mm, rotated rx 180 ry 0 rz -90 deg; joints [34.362, -75.805, -81.797, -22.397, 55.638, -90]
  MoveL 997 to (-446.65, -333.14, 848) mm, rotated rx 180 ry 0 rz -90 deg; joints [34.509, -74.497, -84.484, -21.02, 55.491, -90]
  MoveL 998 to (-450.33, -322.49, 855) mm, rotated rx 180 ry 0 rz -90 deg; joints [34.726, -72.946, -87.192, -19.861, 55.274, -90]
  MoveL 999 to (-456.13, -313.06, 866) mm, rotated rx 180 ry 0 rz -90 deg; joints [35.098, -70.863, -89.993, -19.144, 54.902, -90]
  MoveL 1000 to (-450.86, -296.02, 856) mm, rotated rx 180 ry 0 rz -90 deg; joints [34.758, -71.689, -92.08, -16.231, 55.242, -90]
  MoveL 1001 to (-452.97, -283.92, 860) mm, rotated rx 180 ry 0 rz -90 deg; joints [34.89, -70.636, -94.585, -14.78, 55.11, -90]
  MoveL 1002 to (-455.6, -272, 865) mm, rotated rx 180 ry 0 rz -90 deg; joints [35.063, -69.462, -97.105, -13.433, 54.937, -90]
  MoveL 1003 to (-461.92, -262.02, 877) mm, rotated rx 180 ry 0 rz -90 deg; joints [35.513, -67.254, -99.903, -12.843, 54.487, -90]
  MoveL 1004 to (-464.03, -249.4, 881) mm, rotated rx 180 ry 0 rz -90 deg; joints [35.676, -66.247, -102.355, -11.399, 54.324, -90]
  MoveL 1005 to (-464.55, -235.85, 882) mm, rotated rx 180 ry 0 rz -90 deg; joints [35.718, -65.741, -104.646, -9.613, 54.282, -90]
  MoveL 1006 to (-472.98, -226.05, 898) mm, rotated rx 180 ry 0 rz -90 deg; joints [36.457, -62.841, -107.616, -9.543, 53.543, -90]
  MoveL 1007 to (-471.93, -211.5, 896) mm, rotated rx 180 ry 0 rz -90 deg; joints [36.357, -62.877, -109.746, -7.377, 53.643, -90]
  MoveL 1008 to (-465.61, -194.8, 884) mm, rotated rx 180 ry 0 rz -90 deg; joints [35.803, -64.711, -111.244, -4.045, 54.197, -90]
  MoveL 1009 to (-468.24, -181.96, 889) mm, rotated rx 180 ry 0 rz -90 deg; joints [36.025, -63.726, -113.642, -2.632, 53.975, -90]
  MoveL 1010 to (-466.13, -167.27, 885) mm, rotated rx 180 ry 0 rz -90 deg; joints [35.847, -64.386, -115.441, -0.173, 54.153, -90]
  MoveL 1011 to (-468.24, -154.08, 889) mm, rotated rx 180 ry 0 rz -90 deg; joints [36.025, -63.682, -117.737, 1.418, 53.975, -90]
  MoveL 1012 to (-476.67, -142.66, 905) mm, rotated rx 180 ry 0 rz -90 deg; joints [36.827, -60.729, -120.865, 1.595, 53.173, -90]
  MoveL 1013 to (-468.24, -126.2, 889) mm, rotated rx 180 ry 0 rz -90 deg; joints [36.025, -63.948, -121.677, 5.625, 53.975, -90]
  MoveL 1014 to (-472.46, -113.27, 897) mm, rotated rx 180 ry 0 rz -90 deg; joints [36.407, -62.629, -124.249, 6.879, 53.593, -90]
  MoveL 1015 to (-460.87, -96.77, 875) mm, rotated rx 180 ry 0 rz -90 deg; joints [35.434, -67.319, -124.177, 11.496, 54.566, -90]
  MoveL 1016 to (-461.92, -83.24, 877) mm, rotated rx 180 ry 0 rz -90 deg; joints [35.513, -67.419, -126.144, 13.562, 54.487, -90]
  MoveL 1017 to (-460.87, -69.33, 875) mm, rotated rx 180 ry 0 rz -90 deg; joints [35.434, -68.408, -127.672, 16.08, 54.566, -90]
  MoveL 1018 to (-454.55, -54.84, 863) mm, rotated rx 180 ry 0 rz -90 deg; joints [34.993, -71.487, -128.016, 19.502, 55.007, -90]
  MoveL 1019 to (-454.55, -41.31, 863) mm, rotated rx 180 ry 0 rz -90 deg; joints [34.993, -72.315, -129.598, 21.913, 55.007, -90]
  MoveL 1020 to (-454.55, -27.78, 863) mm, rotated rx 180 ry 0 rz -90 deg; joints [34.993, -73.256, -131.134, 24.39, 55.007, -90]
  MoveL 1021 to (-448.23, -14.05, 851) mm, rotated rx 180 ry 0 rz -90 deg; joints [34.6, -76.618, -131.056, 27.674, 55.4, -90]
  MoveL 1022 to (-445.59, -0.7, 846) mm, rotated rx 180 ry 0 rz -90 deg; joints [34.449, -78.711, -131.748, 30.458, 55.551, -90]
  MoveL 1023 to (-442.96, 12.49, 841) mm, rotated rx 180 ry 0 rz -90 deg; joints [34.305, -80.882, -132.334, 33.216, 55.695, -90]
  MoveL 1024 to (-436.11, 25.28, 828) mm, rotated rx 180 ry 0 rz -90 deg; joints [33.958, -84.478, -131.612, 36.09, 56.042, -90]
  MoveL 1025 to (-435.59, 38.22, 827) mm, rotated rx 180 ry 0 rz -90 deg; joints [33.933, -86.074, -132.572, 38.646, 56.067, -90]
  MoveL 1026 to (-434.01, 51.01, 824) mm, rotated rx 180 ry 0 rz -90 deg; joints [33.859, -88.079, -133.146, 41.224, 56.141, -90]
  MoveL 1027 to (-427.69, 63, 812) mm, rotated rx 180 ry 0 rz -90 deg; joints [33.579, -91.459, -132.157, 43.616, 56.421, -90]
  MoveL 1028 to (-427.16, 75.64, 811) mm, rotated rx 180 ry 0 rz -90 deg; joints [33.557, -93.241, -132.867, 46.108, 56.443, -90]
  MoveL 1029 to (-424.53, 87.81, 806) mm, rotated rx 180 ry 0 rz -90 deg; joints [33.449, -95.612, -132.823, 48.436, 56.551, -90]
  MoveL 1030 to (-419.78, 99.33, 797) mm, rotated rx 180 ry 0 rz -90 deg; joints [33.265, -98.454, -131.989, 50.442, 56.735, -90]
  MoveL 1031 to (-419.78, 111.83, 797) mm, rotated rx 180 ry 0 rz -90 deg; joints [33.265, -100.241, -132.636, 52.878, 56.735, -90]
  MoveL 1032 to (-434.37, -493.88, 850) mm, rotated rx 180 ry 0 rz -90 deg; joints [37.028, -87.988, -45.164, -46.848, 52.972, -90]
  MoveL 1033 to (-440.5, -487.34, 862) mm, rotated rx 180 ry 0 rz -90 deg; joints [37.586, -85.295, -48.993, -45.713, 52.414, -90]
  MoveL 1034 to (-435.9, -468.87, 853) mm, rotated rx 180 ry 0 rz -90 deg; joints [37.162, -84.42, -53.491, -42.088, 52.838, -90]
  MoveL 1035 to (-433.86, -453.36, 849) mm, rotated rx 180 ry 0 rz -90 deg; joints [36.985, -83.356, -57.38, -39.264, 53.015, -90]
  MoveL 1036 to (-434.37, -440.56, 850) mm, rotated rx 180 ry 0 rz -90 deg; joints [37.028, -81.967, -60.902, -37.131, 52.972, -90]
  MoveL 1037 to (-434.37, -427.23, 850) mm, rotated rx 180 ry 0 rz -90 deg; joints [37.028, -80.776, -64.261, -34.963, 52.972, -90]
  MoveL 1038 to (-433.86, -413.42, 849) mm, rotated rx 180 ry 0 rz -90 deg; joints [36.985, -79.784, -67.463, -32.752, 53.015, -90]
  MoveL 1039 to (-436.42, -402.46, 854) mm, rotated rx 180 ry 0 rz -90 deg; joints [37.207, -78.217, -70.535, -31.248, 52.793, -90]
  MoveL 1040 to (-436.93, -389.53, 855) mm, rotated rx 180 ry 0 rz -90 deg; joints [37.253, -77.146, -73.507, -29.347, 52.747, -90]
  MoveL 1041 to (-434.88, -374.36, 851) mm, rotated rx 180 ry 0 rz -90 deg; joints [37.073, -76.734, -76.317, -26.949, 52.927, -90]
  MoveL 1042 to (-438.46, -363.98, 858) mm, rotated rx 180 ry 0 rz -90 deg; joints [37.393, -75.066, -79.184, -25.75, 52.607, -90]
  MoveL 1043 to (-431.3, -344.81, 844) mm, rotated rx 180 ry 0 rz -90 deg; joints [36.772, -76.078, -81.538, -22.384, 53.228, -90]
  MoveL 1044 to (-434.37, -333.93, 850) mm, rotated rx 180 ry 0 rz -90 deg; joints [37.028, -74.631, -84.268, -21.101, 52.972, -90]
  MoveL 1045 to (-439.48, -324.37, 860) mm, rotated rx 180 ry 0 rz -90 deg; joints [37.488, -72.666, -87.084, -20.25, 52.512, -90]
  MoveL 1046 to (-445.1, -314.86, 871) mm, rotated rx 180 ry 0 rz -90 deg; joints [38.048, -70.555, -89.905, -19.54, 51.952, -90]
  MoveL 1047 to (-439.99, -297.75, 861) mm, rotated rx 180 ry 0 rz -90 deg; joints [37.537, -71.378, -92.017, -16.605, 52.463, -90]
  MoveL 1048 to (-445.61, -287.88, 872) mm, rotated rx 180 ry 0 rz -90 deg; joints [38.102, -69.292, -94.812, -15.896, 51.898, -90]
  MoveL 1049 to (-447.15, -275.15, 875) mm, rotated rx 180 ry 0 rz -90 deg; joints [38.267, -68.368, -97.287, -14.345, 51.733, -90]
  MoveL 1050 to (-453.79, -265.31, 888) mm, rotated rx 180 ry 0 rz -90 deg; joints [39.046, -65.953, -100.136, -13.911, 50.954, -90]
  MoveL 1051 to (-453.79, -251.38, 888) mm, rotated rx 180 ry 0 rz -90 deg; joints [39.046, -65.523, -102.456, -12.021, 50.954, -90]
  MoveL 1052 to (-453.79, -237.46, 888) mm, rotated rx 180 ry 0 rz -90 deg; joints [39.046, -65.152, -104.728, -10.12, 50.954, -90]
  MoveL 1053 to (-458.9, -226.05, 898) mm, rotated rx 180 ry 0 rz -90 deg; joints [39.727, -63.185, -107.443, -9.372, 50.273, -90]
  MoveL 1054 to (-459.41, -212.21, 899) mm, rotated rx 180 ry 0 rz -90 deg; joints [39.8, -62.722, -109.72, -7.559, 50.2, -90]
  MoveL 1055 to (-451.75, -194.8, 884) mm, rotated rx 180 ry 0 rz -90 deg; joints [38.795, -65.102, -111.033, -3.865, 51.205, -90]
  MoveL 1056 to (-460.94, -184.62, 902) mm, rotated rx 180 ry 0 rz -90 deg; joints [40.023, -61.782, -114.231, -3.987, 49.977, -90]
  MoveL 1057 to (-457.37, -169.16, 895) mm, rotated rx 180 ry 0 rz -90 deg; joints [39.514, -62.963, -115.905, -1.132, 50.486, -90]
  MoveL 1058 to (-456.35, -154.77, 893) mm, rotated rx 180 ry 0 rz -90 deg; joints [39.377, -63.334, -117.815, 1.149, 50.623, -90]
  MoveL 1059 to (-460.43, -142.03, 901) mm, rotated rx 180 ry 0 rz -90 deg; joints [39.947, -61.873, -120.409, 2.282, 50.053, -90]
  MoveL 1060 to (-455.32, -126.48, 891) mm, rotated rx 180 ry 0 rz -90 deg; joints [39.242, -63.972, -121.623, 5.595, 50.758, -90]
  MoveL 1061 to (-458.9, -113.4, 898) mm, rotated rx 180 ry 0 rz -90 deg; joints [39.727, -62.83, -124.131, 6.96, 50.273, -90]
  MoveL 1062 to (-456.35, -98.76, 893) mm, rotated rx 180 ry 0 rz -90 deg; joints [39.377, -64.18, -125.6, 9.779, 50.623, -90]
  MoveL 1063 to (-451.23, -83.81, 883) mm, rotated rx 180 ry 0 rz -90 deg; joints [38.734, -66.67, -126.482, 13.152, 51.267, -90]
  MoveL 1064 to (-450.21, -69.8, 881) mm, rotated rx 180 ry 0 rz -90 deg; joints [38.613, -67.66, -128.033, 15.693, 51.387, -90]
  MoveL 1065 to (-447.15, -55.61, 875) mm, rotated rx 180 ry 0 rz -90 deg; joints [38.267, -69.579, -129.077, 18.656, 51.733, -90]
  MoveL 1066 to (-442.04, -41.41, 865) mm, rotated rx 180 ry 0 rz -90 deg; joints [37.735, -72.404, -129.525, 21.929, 52.265, -90]
  MoveL 1067 to (-439.99, -27.71, 861) mm, rotated rx 180 ry 0 rz -90 deg; joints [37.537, -74.134, -130.56, 24.694, 52.463, -90]
  MoveL 1068 to (-434.37, -14.03, 850) mm, rotated rx 180 ry 0 rz -90 deg; joints [37.028, -77.297, -130.567, 27.865, 52.972, -90]
  MoveL 1069 to (-436.93, -0.71, 855) mm, rotated rx 180 ry 0 rz -90 deg; joints [37.253, -77.523, -132.627, 30.15, 52.747, -90]
  MoveL 1070 to (-431.3, 12.54, 844) mm, rotated rx 180 ry 0 rz -90 deg; joints [36.772, -80.832, -132.382, 33.214, 53.228, -90]
  MoveL 1071 to (-426.19, 25.47, 834) mm, rotated rx 180 ry 0 rz -90 deg; joints [36.373, -83.944, -132.107, 36.051, 53.627, -90]
  MoveL 1072 to (-424.66, 38.41, 831) mm, rotated rx 180 ry 0 rz -90 deg; joints [36.26, -85.892, -132.771, 38.663, 53.74, -90]
  MoveL 1073 to (-420.06, 50.88, 822) mm, rotated rx 180 ry 0 rz -90 deg; joints [35.937, -88.846, -132.384, 41.23, 54.063, -90]
  MoveL 1074 to (-417.51, 63.38, 817) mm, rotated rx 180 ry 0 rz -90 deg; joints [35.767, -91.18, -132.524, 43.704, 54.233, -90]
  MoveL 1075 to (-412.91, 75.36, 808) mm, rotated rx 180 ry 0 rz -90 deg; joints [35.478, -94.078, -131.889, 45.966, 54.522, -90]
  MoveL 1076 to (-412.4, 87.92, 807) mm, rotated rx 180 ry 0 rz -90 deg; joints [35.447, -95.899, -132.513, 48.413, 54.553, -90]
  MoveL 1077 to (-408.82, 99.7, 800) mm, rotated rx 180 ry 0 rz -90 deg; joints [35.237, -98.499, -132.018, 50.517, 54.763, -90]
  MoveL 1078 to (-410.35, 112.67, 803) mm, rotated rx 180 ry 0 rz -90 deg; joints [35.326, -99.97, -133.197, 53.167, 54.674, -90]
  MoveL 1079 to (-408.31, 124.64, 799) mm, rotated rx 180 ry 0 rz -90 deg; joints [35.208, -102.269, -133.068, 55.337, 54.792, -90]
  MoveL 1080 to (-425, -498.53, 858) mm, rotated rx 180 ry 0 rz -90 deg; joints [39.844, -87.89, -44.255, -47.855, 50.156, -90]
  MoveL 1081 to (-429.46, -490.16, 867) mm, rotated rx 180 ry 0 rz -90 deg; joints [40.409, -85.372, -48.331, -46.297, 49.591, -90]
  MoveL 1082 to (-425.5, -472.17, 859) mm, rotated rx 180 ry 0 rz -90 deg; joints [39.904, -84.369, -52.883, -42.748, 50.096, -90]
  MoveL 1083 to (-421.04, -453.89, 850) mm, rotated rx 180 ry 0 rz -90 deg; joints [39.379, -83.731, -56.963, -39.305, 50.621, -90]
  MoveL 1084 to (-421.04, -440.56, 850) mm, rotated rx 180 ry 0 rz -90 deg; joints [39.379, -82.432, -60.523, -37.045, 50.621, -90]
  MoveL 1085 to (-429.96, -436.28, 868) mm, rotated rx 180 ry 0 rz -90 deg; joints [40.475, -79.405, -63.685, -36.91, 49.525, -90]
  MoveL 1086 to (-427.48, -420.24, 863) mm, rotated rx 180 ry 0 rz -90 deg; joints [40.152, -78.749, -67.055, -34.196, 49.848, -90]
  MoveL 1087 to (-428.97, -408.12, 866) mm, rotated rx 180 ry 0 rz -90 deg; joints [40.344, -77.348, -70.198, -32.454, 49.656, -90]
  MoveL 1088 to (-427.98, -393.63, 864) mm, rotated rx 180 ry 0 rz -90 deg; joints [40.215, -76.571, -73.23, -30.2, 49.785, -90]
  MoveL 1089 to (-426.49, -378.76, 861) mm, rotated rx 180 ry 0 rz -90 deg; joints [40.027, -76.003, -76.114, -27.883, 49.973, -90]
  MoveL 1090 to (-426, -364.83, 860) mm, rotated rx 180 ry 0 rz -90 deg; joints [39.965, -75.282, -78.897, -25.821, 50.035, -90]
  MoveL 1091 to (-420.05, -346.44, 848) mm, rotated rx 180 ry 0 rz -90 deg; joints [39.268, -76.041, -81.306, -22.653, 50.732, -90]
  MoveL 1092 to (-422.53, -335.11, 853) mm, rotated rx 180 ry 0 rz -90 deg; joints [39.549, -74.713, -84.027, -21.261, 50.451, -90]
  MoveL 1093 to (-431.44, -328.52, 871) mm, rotated rx 180 ry 0 rz -90 deg; joints [40.677, -71.66, -87.085, -21.255, 49.323, -90]
  MoveL 1094 to (-430.45, -314.14, 869) mm, rotated rx 180 ry 0 rz -90 deg; joints [40.542, -71.297, -89.553, -19.15, 49.458, -90]
  MoveL 1095 to (-428.97, -299.48, 866) mm, rotated rx 180 ry 0 rz -90 deg; joints [40.344, -71.148, -91.899, -16.953, 49.656, -90]
  MoveL 1096 to (-435.41, -290.19, 879) mm, rotated rx 180 ry 0 rz -90 deg; joints [41.245, -68.749, -94.784, -16.467, 48.755, -90]
  MoveL 1097 to (-431.44, -273.89, 871) mm, rotated rx 180 ry 0 rz -90 deg; joints [40.677, -69.445, -96.832, -13.723, 49.323, -90]
  MoveL 1098 to (-438.87, -264.71, 886) mm, rotated rx 180 ry 0 rz -90 deg; joints [41.782, -66.73, -99.796, -13.474, 48.218, -90]
  MoveL 1099 to (-436.4, -249.4, 881) mm, rotated rx 180 ry 0 rz -90 deg; joints [41.394, -67.105, -101.872, -11.023, 48.606, -90]
  MoveL 1100 to (-444.82, -240.13, 898) mm, rotated rx 180 ry 0 rz -90 deg; joints [42.803, -64.01, -104.933, -11.057, 47.197, -90]
  MoveL 1101 to (-449.77, -228.57, 908) mm, rotated rx 180 ry 0 rz -90 deg; joints [43.77, -61.981, -107.665, -10.354, 46.23, -90]
  MoveL 1102 to (-446.3, -212.68, 901) mm, rotated rx 180 ry 0 rz -90 deg; joints [43.081, -62.863, -109.579, -7.558, 46.919, -90]
  MoveL 1103 to (-442.34, -196.79, 893) mm, rotated rx 180 ry 0 rz -90 deg; joints [42.361, -64.041, -111.308, -4.65, 47.639, -90]
  MoveL 1104 to (-446.3, -184.42, 901) mm, rotated rx 180 ry 0 rz -90 deg; joints [43.081, -62.464, -113.925, -3.611, 46.919, -90]
  MoveL 1105 to (-450.27, -171.8, 909) mm, rotated rx 180 ry 0 rz -90 deg; joints [43.873, -60.868, -116.544, -2.587, 46.127, -90]
  MoveL 1106 to (-446.3, -156.16, 901) mm, rotated rx 180 ry 0 rz -90 deg; joints [43.081, -62.347, -118.112, 0.459, 46.919, -90]
  MoveL 1107 to (-444.82, -141.56, 898) mm, rotated rx 180 ry 0 rz -90 deg; joints [42.803, -62.989, -119.922, 2.911, 47.197, -90]
  MoveL 1108 to (-443.83, -127.19, 896) mm, rotated rx 180 ry 0 rz -90 deg; joints [42.623, -63.539, -121.743, 5.283, 47.377, -90]
  MoveL 1109 to (-446.3, -113.77, 901) mm, rotated rx 180 ry 0 rz -90 deg; joints [43.081, -62.774, -124.103, 6.877, 46.919, -90]
  MoveL 1110 to (-441.35, -98.54, 891) mm, rotated rx 180 ry 0 rz -90 deg; joints [42.19, -65.156, -125.116, 10.272, 47.81, -90]
  MoveL 1111 to (-443.33, -84.95, 895) mm, rotated rx 180 ry 0 rz -90 deg; joints [42.535, -64.786, -127.336, 12.122, 47.466, -90]
  MoveL 1112 to (-436.4, -69.8, 881) mm, rotated rx 180 ry 0 rz -90 deg; joints [41.394, -68.25, -127.693, 15.942, 48.606, -90]
  MoveL 1113 to (-432.93, -55.54, 874) mm, rotated rx 180 ry 0 rz -90 deg; joints [40.884, -70.377, -128.601, 18.978, 49.116, -90]
  MoveL 1114 to (-428.47, -41.41, 865) mm, rotated rx 180 ry 0 rz -90 deg; joints [40.279, -73.002, -129.135, 22.137, 49.721, -90]
  MoveL 1115 to (-428.97, -27.87, 866) mm, rotated rx 180 ry 0 rz -90 deg; joints [40.344, -73.75, -130.791, 24.541, 49.656, -90]
  MoveL 1116 to (-422.53, -14.08, 853) mm, rotated rx 180 ry 0 rz -90 deg; joints [39.549, -77.323, -130.54, 27.863, 50.451, -90]
  MoveL 1117 to (-421.54, -0.7, 851) mm, rotated rx 180 ry 0 rz -90 deg; joints [39.435, -78.863, -131.632, 30.495, 50.565, -90]
  MoveL 1118 to (-419.06, 12.57, 846) mm, rotated rx 180 ry 0 rz -90 deg; joints [39.159, -81.051, -132.213, 33.263, 50.841, -90]
  MoveL 1119 to (-414.11, 25.53, 836) mm, rotated rx 180 ry 0 rz -90 deg; joints [38.64, -84.164, -131.928, 36.092, 51.36, -90]
  MoveL 1120 to (-413.12, 38.55, 834) mm, rotated rx 180 ry 0 rz -90 deg; joints [38.542, -85.949, -132.745, 38.694, 51.458, -90]
  MoveL 1121 to (-407.17, 50.88, 822) mm, rotated rx 180 ry 0 rz -90 deg; joints [37.983, -89.374, -131.868, 41.242, 52.017, -90]
  MoveL 1122 to (-405.19, 63.46, 818) mm, rotated rx 180 ry 0 rz -90 deg; joints [37.808, -91.545, -132.162, 43.707, 52.192, -90]
  MoveL 1123 to (-397.76, 74.89, 803) mm, rotated rx 180 ry 0 rz -90 deg; joints [37.198, -95.232, -130.491, 45.723, 52.802, -90]
  MoveL 1124 to (-402.71, 88.57, 813) mm, rotated rx 180 ry 0 rz -90 deg; joints [37.597, -95.606, -132.999, 48.605, 52.403, -90]
  MoveL 1125 to (-398.26, 100.2, 804) mm, rotated rx 180 ry 0 rz -90 deg; joints [37.236, -98.479, -132.158, 50.637, 52.764, -90]
  MoveL 1126 to (-398.26, 112.81, 804) mm, rotated rx 180 ry 0 rz -90 deg; joints [37.236, -100.292, -132.808, 53.1, 52.764, -90]
  MoveL 1127 to (-394.79, 124.32, 797) mm, rotated rx 180 ry 0 rz -90 deg; joints [36.972, -102.873, -132.134, 55.008, 53.028, -90]
  MoveL 1128 to (-416.83, -504.92, 869) mm, rotated rx 180 ry 0 rz -90 deg; joints [43.003, -87.682, -43.039, -49.279, 46.997, -90]
  MoveL 1129 to (-413.95, -487.9, 863) mm, rotated rx 180 ry 0 rz -90 deg; joints [42.539, -86.236, -48.041, -45.723, 47.461, -90]
  MoveL 1130 to (-412.03, -472.17, 859) mm, rotated rx 180 ry 0 rz -90 deg; joints [42.244, -84.917, -52.41, -42.673, 47.756, -90]
  MoveL 1131 to (-410.11, -456.56, 855) mm, rotated rx 180 ry 0 rz -90 deg; joints [41.959, -83.809, -56.392, -39.799, 48.041, -90]
  MoveL 1132 to (-412.03, -445.23, 859) mm, rotated rx 180 ry 0 rz -90 deg; joints [42.244, -82.088, -59.945, -37.967, 47.756, -90]
  MoveL 1133 to (-411.55, -431.26, 858) mm, rotated rx 180 ry 0 rz -90 deg; joints [42.172, -80.953, -63.402, -35.645, 47.828, -90]
  MoveL 1134 to (-415.87, -422.18, 867) mm, rotated rx 180 ry 0 rz -90 deg; joints [42.845, -78.859, -66.629, -34.512, 47.155, -90]
  MoveL 1135 to (-418.27, -410.94, 872) mm, rotated rx 180 ry 0 rz -90 deg; joints [43.244, -77.222, -69.797, -32.981, 46.756, -90]
  MoveL 1136 to (-419.7, -398.64, 875) mm, rotated rx 180 ry 0 rz -90 deg; joints [43.493, -75.852, -72.882, -31.267, 46.507, -90]
  MoveL 1137 to (-412.51, -364.83, 860) mm, rotated rx 180 ry 0 rz -90 deg; joints [42.317, -75.827, -78.515, -25.658, 47.683, -90]
  MoveL 1138 to (-408.67, -348.08, 852) mm, rotated rx 180 ry 0 rz -90 deg; joints [41.752, -76.08, -81.019, -22.901, 48.248, -90]
  MoveL 1139 to (-418.27, -342.57, 872) mm, rotated rx 180 ry 0 rz -90 deg; joints [43.244, -72.776, -84.153, -23.072, 46.756, -90]
  MoveL 1140 to (-424.02, -333.43, 884) mm, rotated rx 180 ry 0 rz -90 deg; joints [44.286, -70.473, -87.052, -22.476, 45.714, -90]
  MoveL 1141 to (-418.74, -315.59, 873) mm, rotated rx 180 ry 0 rz -90 deg; joints [43.327, -71.304, -89.325, -19.371, 46.673, -90]
  MoveL 1142 to (-419.22, -302.24, 874) mm, rotated rx 180 ry 0 rz -90 deg; joints [43.41, -70.578, -91.834, -17.588, 46.59, -90]
  MoveL 1143 to (-425.94, -293.16, 888) mm, rotated rx 180 ry 0 rz -90 deg; joints [44.663, -68.005, -94.765, -17.23, 45.337, -90]
  MoveL 1144 to (-420.66, -275.77, 877) mm, rotated rx 180 ry 0 rz -90 deg; joints [43.664, -69.126, -96.741, -14.133, 46.337, -90]
  MoveL 1145 to (-429.3, -267.4, 895) mm, rotated rx 180 ry 0 rz -90 deg; joints [45.362, -65.924, -99.837, -14.239, 44.638, -90]
  MoveL 1146 to (-424.02, -250.25, 884) mm, rotated rx 180 ry 0 rz -90 deg; joints [44.286, -67.224, -101.677, -11.099, 45.714, -90]
  MoveL 1147 to (-429.78, -239.6, 896) mm, rotated rx 180 ry 0 rz -90 deg; joints [45.466, -64.934, -104.527, -10.539, 44.534, -90]
  MoveL 1148 to (-431.7, -226.55, 900) mm, rotated rx 180 ry 0 rz -90 deg; joints [45.895, -63.935, -106.985, -9.08, 44.105, -90]
  MoveL 1149 to (-435.53, -214.33, 908) mm, rotated rx 180 ry 0 rz -90 deg; joints [46.814, -62.265, -109.633, -8.103, 43.186, -90]
  MoveL 1150 to (-433.61, -199.21, 904) mm, rotated rx 180 ry 0 rz -90 deg; joints [46.344, -62.724, -111.629, -5.647, 43.657, -90]
  MoveL 1151 to (-434.57, -185.44, 906) mm, rotated rx 180 ry 0 rz -90 deg; joints [46.576, -62.19, -113.911, -3.898, 43.424, -90]
  MoveL 1152 to (-434.57, -171.24, 906) mm, rotated rx 180 ry 0 rz -90 deg; joints [46.576, -62.084, -116.041, -1.875, 43.424, -90]
  MoveL 1153 to (-438.89, -158.59, 915) mm, rotated rx 180 ry 0 rz -90 deg; joints [47.694, -60.304, -118.739, -0.957, 42.306, -90]
  MoveL 1154 to (-432.66, -142.19, 902) mm, rotated rx 180 ry 0 rz -90 deg; joints [46.116, -62.885, -119.882, 2.768, 43.884, -90]
  MoveL 1155 to (-431.7, -127.76, 900) mm, rotated rx 180 ry 0 rz -90 deg; joints [45.895, -63.433, -121.715, 5.148, 44.105, -90]
  MoveL 1156 to (-430.74, -113.4, 898) mm, rotated rx 180 ry 0 rz -90 deg; joints [45.678, -64.085, -123.488, 7.573, 44.322, -90]
  MoveL 1157 to (-430.26, -99.2, 897) mm, rotated rx 180 ry 0 rz -90 deg; joints [45.571, -64.639, -125.293, 9.932, 44.429, -90]
  MoveL 1158 to (-428.34, -84.76, 893) mm, rotated rx 180 ry 0 rz -90 deg; joints [45.156, -65.922, -126.754, 12.676, 44.844, -90]
  MoveL 1159 to (-425.46, -70.28, 887) mm, rotated rx 180 ry 0 rz -90 deg; joints [44.567, -67.74, -127.915, 15.655, 45.433, -90]
  MoveL 1160 to (-424.5, -56.24, 885) mm, rotated rx 180 ry 0 rz -90 deg; joints [44.379, -68.853, -129.411, 18.264, 45.621, -90]
  MoveL 1161 to (-415.39, -41.46, 866) mm, rotated rx 180 ry 0 rz -90 deg; joints [42.768, -73.511, -128.79, 22.301, 47.233, -90]
  MoveL 1162 to (-416.35, -27.94, 868) mm, rotated rx 180 ry 0 rz -90 deg; joints [42.924, -74.066, -130.569, 24.635, 47.076, -90]
  MoveL 1163 to (-413.95, -14.25, 863) mm, rotated rx 180 ry 0 rz -90 deg; joints [42.539, -76.108, -131.387, 27.495, 47.461, -90]
  MoveL 1164 to (-403.88, -0.7, 842) mm, rotated rx 180 ry 0 rz -90 deg; joints [41.1, -81.175, -129.826, 31.001, 48.9, -90]
  MoveL 1165 to (-405.79, 12.57, 846) mm, rotated rx 180 ry 0 rz -90 deg; joints [41.354, -81.716, -131.676, 33.393, 48.646, -90]
  MoveL 1166 to (-401.96, 25.59, 838) mm, rotated rx 180 ry 0 rz -90 deg; joints [40.854, -84.466, -131.677, 36.143, 49.146, -90]
  MoveL 1167 to (-401, 38.64, 836) mm, rotated rx 180 ry 0 rz -90 deg; joints [40.734, -86.249, -132.491, 38.74, 49.266, -90]
  MoveL 1168 to (-396.68, 51.19, 827) mm, rotated rx 180 ry 0 rz -90 deg; joints [40.217, -89.204, -132.095, 41.299, 49.783, -90]
  MoveL 1169 to (-396.2, 64.08, 826) mm, rotated rx 180 ry 0 rz -90 deg; joints [40.162, -90.958, -132.894, 43.851, 49.838, -90]
  MoveL 1170 to (-394.28, 76.66, 822) mm, rotated rx 180 ry 0 rz -90 deg; joints [39.945, -93.213, -133.115, 46.327, 50.055, -90]
  MoveL 1171 to (-389.01, 88.35, 811) mm, rotated rx 180 ry 0 rz -90 deg; joints [39.382, -96.388, -132.035, 48.423, 50.618, -90]
  MoveL 1172 to (-388.05, 100.82, 809) mm, rotated rx 180 ry 0 rz -90 deg; joints [39.285, -98.393, -132.408, 50.802, 50.715, -90]
  MoveL 1173 to (-386.61, 113.09, 806) mm, rotated rx 180 ry 0 rz -90 deg; joints [39.141, -100.554, -132.529, 53.082, 50.859, -90]
  MoveL 1174 to (-384.21, 124.95, 801) mm, rotated rx 180 ry 0 rz -90 deg; joints [38.909, -102.931, -132.211, 55.142, 51.091, -90]
  MoveL 1175 to (-401.81, -503.18, 866) mm, rotated rx 180 ry 0 rz -90 deg; joints [45.056, -88.551, -42.606, -48.843, 44.944, -90]
  MoveL 1176 to (-403.2, -491.29, 869) mm, rotated rx 180 ry 0 rz -90 deg; joints [45.323, -86.408, -47.172, -46.42, 44.677, -90]
  MoveL 1177 to (-399.49, -473.27, 861) mm, rotated rx 180 ry 0 rz -90 deg; joints [44.626, -85.376, -51.79, -42.834, 45.374, -90]
  MoveL 1178 to (-398.1, -458.16, 858) mm, rotated rx 180 ry 0 rz -90 deg; joints [44.377, -84.155, -55.792, -40.053, 45.624, -90]
  MoveL 1179 to (-404.59, -451.97, 872) mm, rotated rx 180 ry 0 rz -90 deg; joints [45.598, -81.453, -59.194, -39.353, 44.402, -90]
  MoveL 1180 to (-401.81, -435.28, 866) mm, rotated rx 180 ry 0 rz -90 deg; joints [45.056, -80.753, -62.833, -36.414, 44.944, -90]
  MoveL 1181 to (-403.66, -423.64, 870) mm, rotated rx 180 ry 0 rz -90 deg; joints [45.414, -79.158, -66.146, -34.697, 44.586, -90]
  MoveL 1182 to (-405.98, -412.36, 875) mm, rotated rx 180 ry 0 rz -90 deg; joints [45.881, -77.51, -69.345, -33.146, 44.119, -90]
  MoveL 1183 to (-412.94, -405.47, 890) mm, rotated rx 180 ry 0 rz -90 deg; joints [47.425, -74.784, -72.426, -32.789, 42.575, -90]
  MoveL 1184 to (-404.59, -383.6, 872) mm, rotated rx 180 ry 0 rz -90 deg; joints [45.598, -75.858, -75.413, -28.729, 44.402, -90]
  MoveL 1185 to (-403.2, -368.65, 869) mm, rotated rx 180 ry 0 rz -90 deg; joints [45.323, -75.344, -78.233, -26.423, 44.677, -90]
  MoveL 1186 to (-406.91, -358.29, 877) mm, rotated rx 180 ry 0 rz -90 deg; joints [46.074, -73.532, -81.141, -25.327, 43.926, -90]
  MoveL 1187 to (-403.2, -341.39, 869) mm, rotated rx 180 ry 0 rz -90 deg; joints [45.323, -73.803, -83.66, -22.538, 44.677, -90]
  MoveL 1188 to (-409.69, -333.05, 883) mm, rotated rx 180 ry 0 rz -90 deg; joints [46.676, -71.249, -86.633, -22.118, 43.324, -90]
  MoveL 1189 to (-410.16, -319.56, 884) mm, rotated rx 180 ry 0 rz -90 deg; joints [46.78, -70.437, -89.247, -20.316, 43.22, -90]
  MoveL 1190 to (-409.69, -305.35, 883) mm, rotated rx 180 ry 0 rz -90 deg; joints [46.676, -69.959, -91.738, -18.303, 43.324, -90]
  MoveL 1191 to (-410.62, -292.17, 885) mm, rotated rx 180 ry 0 rz -90 deg; joints [46.885, -69.111, -94.268, -16.622, 43.115, -90]
  MoveL 1192 to (-409.23, -277.35, 882) mm, rotated rx 180 ry 0 rz -90 deg; joints [46.573, -69.052, -96.549, -14.4, 43.427, -90]
  MoveL 1193 to (-416.65, -268.3, 898) mm, rotated rx 180 ry 0 rz -90 deg; joints [48.35, -66.151, -99.578, -14.271, 41.65, -90]
  MoveL 1194 to (-417.58, -254.78, 900) mm, rotated rx 180 ry 0 rz -90 deg; joints [48.594, -65.389, -102.021, -12.59, 41.406, -90]
  MoveL 1195 to (-426.86, -246.02, 920) mm, rotated rx 180 ry 0 rz -90 deg; joints [51.364, -61.704, -105.195, -13.101, 38.636, -90]
  MoveL 1196 to (-420.37, -228.06, 906) mm, rotated rx 180 ry 0 rz -90 deg; joints [49.359, -63.654, -106.907, -9.439, 40.641, -90]
  MoveL 1197 to (-423.15, -215.27, 912) mm, rotated rx 180 ry 0 rz -90 deg; joints [50.177, -62.316, -109.469, -8.216, 39.823, -90]
  MoveL 1198 to (-425.93, -202.29, 918) mm, rotated rx 180 ry 0 rz -90 deg; joints [51.057, -60.977, -112.024, -6.998, 38.944, -90]
  MoveL 1199 to (-429.18, -189.33, 925) mm, rotated rx 180 ry 0 rz -90 deg; joints [52.168, -59.449, -114.63, -5.921, 37.832, -90]
  MoveL 1200 to (-423.61, -172.56, 913) mm, rotated rx 180 ry 0 rz -90 deg; joints [50.32, -61.557, -116.105, -2.338, 39.68, -90]
  MoveL 1201 to (-424.54, -158.59, 915) mm, rotated rx 180 ry 0 rz -90 deg; joints [50.609, -61.119, -118.356, -0.525, 39.391, -90]
  MoveL 1202 to (-420.37, -142.82, 906) mm, rotated rx 180 ry 0 rz -90 deg; joints [49.359, -62.917, -119.774, 2.691, 40.641, -90]
  MoveL 1203 to (-420.83, -128.76, 907) mm, rotated rx 180 ry 0 rz -90 deg; joints [49.491, -62.864, -121.859, 4.723, 40.509, -90]
  MoveL 1204 to (-419.44, -114.15, 904) mm, rotated rx 180 ry 0 rz -90 deg; joints [49.098, -63.707, -123.572, 7.28, 40.902, -90]
  MoveL 1205 to (-413.41, -98.54, 891) mm, rotated rx 180 ry 0 rz -90 deg; joints [47.537, -66.696, -124.268, 10.964, 42.463, -90]
  MoveL 1206 to (-416.65, -85.23, 898) mm, rotated rx 180 ry 0 rz -90 deg; joints [48.35, -65.742, -126.781, 12.523, 41.65, -90]
  MoveL 1207 to (-411.55, -70.28, 887) mm, rotated rx 180 ry 0 rz -90 deg; joints [47.098, -68.586, -127.423, 16.01, 42.902, -90]
  MoveL 1208 to (-408.77, -55.99, 881) mm, rotated rx 180 ry 0 rz -90 deg; joints [46.471, -70.515, -128.447, 18.963, 43.529, -90]
  MoveL 1209 to (-404.59, -41.74, 872) mm, rotated rx 180 ry 0 rz -90 deg; joints [45.598, -73.145, -128.987, 22.133, 44.402, -90]
  MoveL 1210 to (-404.13, -28.04, 871) mm, rotated rx 180 ry 0 rz -90 deg; joints [45.506, -74.294, -130.4, 24.694, 44.494, -90]
  MoveL 1211 to (-401.81, -14.29, 866) mm, rotated rx 180 ry 0 rz -90 deg; joints [45.056, -76.335, -131.218, 27.553, 44.944, -90]
  MoveL 1212 to (-395.31, -0.7, 852) mm, rotated rx 180 ry 0 rz -90 deg; joints [43.897, -80.127, -130.658, 30.785, 46.103, -90]
  MoveL 1213 to (-392.99, 12.58, 847) mm, rotated rx 180 ry 0 rz -90 deg; joints [43.516, -82.286, -131.212, 33.498, 46.484, -90]
  MoveL 1214 to (-388.82, 25.59, 838) mm, rotated rx 180 ry 0 rz -90 deg; joints [42.868, -85.182, -131.048, 36.23, 47.132, -90]
  MoveL 1215 to (-385.57, 38.41, 831) mm, rotated rx 180 ry 0 rz -90 deg; joints [42.396, -87.747, -131.058, 38.806, 47.604, -90]
  MoveL 1216 to (-384.18, 51.25, 828) mm, rotated rx 180 ry 0 rz -90 deg; joints [42.201, -89.716, -131.602, 41.318, 47.8, -90]
  MoveL 1217 to (-383.25, 64.08, 826) mm, rotated rx 180 ry 0 rz -90 deg; joints [42.073, -91.602, -132.228, 43.83, 47.927, -90]
  MoveL 1218 to (-384.18, 77.22, 828) mm, rotated rx 180 ry 0 rz -90 deg; joints [42.201, -93.01, -133.453, 46.463, 47.8, -90]
  MoveL 1219 to (-379.07, 89.01, 817) mm, rotated rx 180 ry 0 rz -90 deg; joints [41.522, -96.213, -132.386, 48.599, 48.478, -90]
  MoveL 1220 to (-375.82, 100.95, 810) mm, rotated rx 180 ry 0 rz -90 deg; joints [41.119, -98.829, -131.89, 50.719, 48.881, -90]
  MoveL 1221 to (-375.82, 113.65, 810) mm, rotated rx 180 ry 0 rz -90 deg; joints [41.119, -100.65, -132.537, 53.187, 48.881, -90]
  MoveL 1222 to (-375.67, -486.91, 838) mm, rotated rx 180 ry 0 rz -90 deg; joints [44.784, -91.42, -43.227, -45.352, 45.216, -90]
  MoveL 1223 to (-393.61, -496.38, 878) mm, rotated rx 180 ry 0 rz -90 deg; joints [48.44, -86.455, -46.041, -47.504, 41.56, -90]
  MoveL 1224 to (-392.26, -480.96, 875) mm, rotated rx 180 ry 0 rz -90 deg; joints [48.12, -84.908, -50.647, -44.446, 41.88, -90]
  MoveL 1225 to (-392.71, -467.78, 876) mm, rotated rx 180 ry 0 rz -90 deg; joints [48.225, -83.227, -54.713, -42.06, 41.775, -90]
  MoveL 1226 to (-395.4, -457.15, 882) mm, rotated rx 180 ry 0 rz -90 deg; joints [48.88, -81.216, -58.394, -40.389, 41.12, -90]
  MoveL 1227 to (-390.92, -438.29, 872) mm, rotated rx 180 ry 0 rz -90 deg; joints [47.808, -80.847, -62.211, -36.943, 42.192, -90]
  MoveL 1228 to (-391.37, -425.11, 873) mm, rotated rx 180 ry 0 rz -90 deg; joints [47.911, -79.54, -65.597, -34.863, 42.089, -90]
  MoveL 1229 to (-391.37, -411.42, 873) mm, rotated rx 180 ry 0 rz -90 deg; joints [47.911, -78.426, -68.839, -32.735, 42.089, -90]
  MoveL 1230 to (-394.95, -401.37, 881) mm, rotated rx 180 ry 0 rz -90 deg; joints [48.769, -76.495, -71.966, -31.539, 41.231, -90]
  MoveL 1231 to (-393.16, -385.8, 877) mm, rotated rx 180 ry 0 rz -90 deg; joints [48.332, -75.975, -74.964, -29.06, 41.668, -90]
  MoveL 1232 to (-391.37, -370.35, 873) mm, rotated rx 180 ry 0 rz -90 deg; joints [47.911, -75.564, -77.803, -26.633, 42.089, -90]
  MoveL 1233 to (-395.85, -360.74, 883) mm, rotated rx 180 ry 0 rz -90 deg; joints [48.993, -73.499, -80.766, -25.735, 41.007, -90]
  MoveL 1234 to (-387.78, -339.82, 865) mm, rotated rx 180 ry 0 rz -90 deg; joints [47.113, -75.041, -83.058, -21.901, 42.887, -90]
  MoveL 1235 to (-394.95, -332.29, 881) mm, rotated rx 180 ry 0 rz -90 deg; joints [48.769, -72.249, -86.117, -21.634, 41.231, -90]
  MoveL 1236 to (-401.23, -323.54, 895) mm, rotated rx 180 ry 0 rz -90 deg; joints [50.435, -69.678, -89.085, -21.236, 39.565, -90]
  MoveL 1237 to (-399.43, -308.12, 891) mm, rotated rx 180 ry 0 rz -90 deg; joints [49.936, -69.585, -91.538, -18.877, 40.064, -90]
  MoveL 1238 to (-402.57, -296.46, 898) mm, rotated rx 180 ry 0 rz -90 deg; joints [50.824, -67.992, -94.267, -17.741, 39.176, -90]
  MoveL 1239 to (-398.09, -279.23, 888) mm, rotated rx 180 ry 0 rz -90 deg; joints [49.574, -68.929, -96.338, -14.733, 40.426, -90]
  MoveL 1240 to (-403.02, -268.6, 899) mm, rotated rx 180 ry 0 rz -90 deg; joints [50.956, -66.796, -99.176, -14.029, 39.044, -90]
  MoveL 1241 to (-407.95, -257.61, 910) mm, rotated rx 180 ry 0 rz -90 deg; joints [52.505, -64.622, -102.003, -13.374, 37.495, -90]
  MoveL 1242 to (-406.61, -242.54, 907) mm, rotated rx 180 ry 0 rz -90 deg; joints [52.064, -64.686, -104.222, -11.092, 37.936, -90]
  MoveL 1243 to (-410.19, -230.33, 915) mm, rotated rx 180 ry 0 rz -90 deg; joints [53.273, -62.996, -106.904, -10.1, 36.727, -90]
  MoveL 1244 to (-415.13, -218.58, 926) mm, rotated rx 180 ry 0 rz -90 deg; joints [55.129, -60.757, -109.725, -9.519, 34.871, -90]
  MoveL 1245 to (-411.99, -202.51, 919) mm, rotated rx 180 ry 0 rz -90 deg; joints [53.92, -61.704, -111.646, -6.651, 36.08, -90]
  MoveL 1246 to (-416.02, -189.95, 928) mm, rotated rx 180 ry 0 rz -90 deg; joints [55.494, -59.831, -114.368, -5.801, 34.506, -90]
  MoveL 1247 to (-408.85, -172.37, 912) mm, rotated rx 180 ry 0 rz -90 deg; joints [52.807, -62.672, -115.582, -1.746, 37.193, -90]
  MoveL 1248 to (-413.78, -159.97, 923) mm, rotated rx 180 ry 0 rz -90 deg; joints [54.598, -60.524, -118.434, -1.042, 35.402, -90]
  MoveL 1249 to (-408.85, -143.77, 912) mm, rotated rx 180 ry 0 rz -90 deg; joints [52.807, -62.699, -119.746, 2.445, 37.193, -90]
  MoveL 1250 to (-415.57, -131.59, 927) mm, rotated rx 180 ry 0 rz -90 deg; joints [55.31, -59.787, -122.919, 2.705, 34.69, -90]
  MoveL 1251 to (-407.95, -114.91, 910) mm, rotated rx 180 ry 0 rz -90 deg; joints [52.505, -63.472, -123.582, 7.054, 37.495, -90]
  MoveL 1252 to (-401.68, -99.09, 896) mm, rotated rx 180 ry 0 rz -90 deg; joints [50.563, -66.651, -124.211, 10.862, 39.437, -90]
  MoveL 1253 to (-401.68, -85.04, 896) mm, rotated rx 180 ry 0 rz -90 deg; joints [50.563, -67.133, -126.036, 13.169, 39.437, -90]
  MoveL 1254 to (-401.23, -70.91, 895) mm, rotated rx 180 ry 0 rz -90 deg; joints [50.435, -67.925, -127.712, 15.638, 39.565, -90]
  MoveL 1255 to (-394.95, -55.99, 881) mm, rotated rx 180 ry 0 rz -90 deg; joints [48.769, -71.461, -127.855, 19.316, 41.231, -90]
  MoveL 1256 to (-393.61, -42.03, 878) mm, rotated rx 180 ry 0 rz -90 deg; joints [48.44, -72.892, -129.109, 22.001, 41.56, -90]
  MoveL 1257 to (-391.81, -28.13, 874) mm, rotated rx 180 ry 0 rz -90 deg; joints [48.015, -74.631, -130.155, 24.786, 41.985, -90]
  MoveL 1258 to (-391.37, -14.41, 873) mm, rotated rx 180 ry 0 rz -90 deg; joints [47.911, -75.898, -131.508, 27.406, 42.089, -90]
  MoveL 1259 to (-384.64, -0.71, 858) mm, rotated rx 180 ry 0 rz -90 deg; joints [46.459, -79.892, -130.841, 30.733, 43.541, -90]
  MoveL 1260 to (-381.95, 12.66, 852) mm, rotated rx 180 ry 0 rz -90 deg; joints [45.927, -82.238, -131.264, 33.503, 44.073, -90]
  MoveL 1261 to (-377.92, 25.74, 843) mm, rotated rx 180 ry 0 rz -90 deg; joints [45.178, -85.138, -131.114, 36.253, 44.822, -90]
  MoveL 1262 to (-380.61, 39.24, 849) mm, rotated rx 180 ry 0 rz -90 deg; joints [45.672, -85.614, -133.176, 38.79, 44.329, -90]
  MoveL 1263 to (-374.78, 51.75, 836) mm, rotated rx 180 ry 0 rz -90 deg; joints [44.63, -89.235, -132.173, 41.408, 45.37, -90]
  MoveL 1264 to (-368.5, 63.77, 822) mm, rotated rx 180 ry 0 rz -90 deg; joints [43.619, -92.867, -130.826, 43.693, 46.382, -90]
  MoveL 1265 to (-371.19, 77.22, 828) mm, rotated rx 180 ry 0 rz -90 deg; joints [44.039, -93.694, -132.706, 46.4, 45.961, -90]
  MoveL 1266 to (-370.3, 89.99, 826) mm, rotated rx 180 ry 0 rz -90 deg; joints [43.897, -95.721, -133.178, 48.9, 46.103, -90]
  MoveL 1267 to (-362.67, 100.82, 809) mm, rotated rx 180 ry 0 rz -90 deg; joints [42.766, -99.542, -130.954, 50.496, 47.234, -90]
  MoveL 1268 to (-368.05, 115.19, 821) mm, rotated rx 180 ry 0 rz -90 deg; joints [43.55, -100.052, -133.709, 53.761, 46.45, -90]
  MoveL 1269 to (-379.84, -496.38, 878) mm, rotated rx 180 ry 0 rz -90 deg; joints [50.556, -87.276, -45.292, -47.432, 39.444, -90]
  MoveL 1270 to (-380.27, -483.16, 879) mm, rotated rx 180 ry 0 rz -90 deg; joints [50.673, -85.384, -49.781, -44.836, 39.327, -90]
  MoveL 1271 to (-378.97, -467.78, 876) mm, rotated rx 180 ry 0 rz -90 deg; joints [50.326, -84.018, -54.05, -41.932, 39.674, -90]
  MoveL 1272 to (-383.73, -459.74, 887) mm, rotated rx 180 ry 0 rz -90 deg; joints [51.645, -81.547, -57.636, -40.817, 38.355, -90]
  MoveL 1273 to (-383.3, -445.33, 886) mm, rotated rx 180 ry 0 rz -90 deg; joints [51.52, -80.254, -61.372, -38.373, 38.48, -90]
  MoveL 1274 to (-377.68, -425.11, 873) mm, rotated rx 180 ry 0 rz -90 deg; joints [49.988, -80.317, -64.999, -34.684, 40.012, -90]
  MoveL 1275 to (-378.11, -411.89, 874) mm, rotated rx 180 ry 0 rz -90 deg; joints [50.1, -79.096, -68.256, -32.649, 39.9, -90]
  MoveL 1276 to (-383.3, -403.65, 886) mm, rotated rx 180 ry 0 rz -90 deg; joints [51.52, -76.726, -71.412, -31.862, 38.48, -90]
  MoveL 1277 to (-381.14, -387.56, 881) mm, rotated rx 180 ry 0 rz -90 deg; joints [50.91, -76.298, -74.443, -29.259, 39.09, -90]
  MoveL 1278 to (-378.54, -371.19, 875) mm, rotated rx 180 ry 0 rz -90 deg; joints [50.212, -76.11, -77.28, -26.61, 39.788, -90]
  MoveL 1279 to (-382.43, -361.15, 884) mm, rotated rx 180 ry 0 rz -90 deg; joints [51.272, -74.178, -80.248, -25.574, 38.728, -90]
  MoveL 1280 to (-384.16, -348.86, 888) mm, rotated rx 180 ry 0 rz -90 deg; joints [51.772, -72.883, -83.082, -24.035, 38.228, -90]
  MoveL 1281 to (-390.65, -340.59, 903) mm, rotated rx 180 ry 0 rz -90 deg; joints [53.822, -70.183, -86.089, -23.728, 36.178, -90]
  MoveL 1282 to (-392.38, -327.88, 907) mm, rotated rx 180 ry 0 rz -90 deg; joints [54.422, -68.906, -88.857, -22.237, 35.578, -90]
  MoveL 1283 to (-390.22, -311.93, 902) mm, rotated rx 180 ry 0 rz -90 deg; joints [53.676, -68.904, -91.353, -19.743, 36.324, -90]
  MoveL 1284 to (-395.85, -302.07, 915) mm, rotated rx 180 ry 0 rz -90 deg; joints [55.699, -66.43, -94.274, -19.296, 34.301, -90]
  MoveL 1285 to (-391.52, -284.58, 905) mm, rotated rx 180 ry 0 rz -90 deg; joints [54.119, -67.293, -96.479, -16.229, 35.881, -90]
  MoveL 1286 to (-390.22, -269.49, 902) mm, rotated rx 180 ry 0 rz -90 deg; joints [53.676, -67.239, -98.791, -13.97, 36.324, -90]
  MoveL 1287 to (-395.41, -258.74, 914) mm, rotated rx 180 ry 0 rz -90 deg; joints [55.533, -64.931, -101.671, -13.398, 34.467, -90]
  MoveL 1288 to (-397.14, -245.48, 918) mm, rotated rx 180 ry 0 rz -90 deg; joints [56.206, -63.86, -104.213, -11.927, 33.794, -90]
  MoveL 1289 to (-398.87, -232.09, 922) mm, rotated rx 180 ry 0 rz -90 deg; joints [56.909, -62.812, -106.734, -10.453, 33.091, -90]
  MoveL 1290 to (-405.36, -221.17, 937) mm, rotated rx 180 ry 0 rz -90 deg; joints [59.856, -59.879, -109.74, -10.381, 30.144, -90]
  MoveL 1291 to (-402.77, -205.16, 931) mm, rotated rx 180 ry 0 rz -90 deg; joints [58.614, -60.609, -111.775, -7.616, 31.386, -90]
  MoveL 1292 to (-401.04, -189.74, 927) mm, rotated rx 180 ry 0 rz -90 deg; joints [57.834, -61.095, -113.812, -5.093, 32.166, -90]
  MoveL 1293 to (-398.44, -174.07, 921) mm, rotated rx 180 ry 0 rz -90 deg; joints [56.731, -62.06, -115.638, -2.302, 33.269, -90]
  MoveL 1294 to (-400.17, -160.32, 925) mm, rotated rx 180 ry 0 rz -90 deg; joints [57.458, -61.249, -118.04, -0.711, 32.542, -90]
  MoveL 1295 to (-401.04, -146.13, 927) mm, rotated rx 180 ry 0 rz -90 deg; joints [57.834, -60.869, -120.293, 1.162, 32.166, -90]
  MoveL 1296 to (-401.04, -131.59, 927) mm, rotated rx 180 ry 0 rz -90 deg; joints [57.834, -60.959, -122.375, 3.334, 32.166, -90]
  MoveL 1297 to (-395.85, -115.54, 915) mm, rotated rx 180 ry 0 rz -90 deg; joints [55.699, -63.588, -123.43, 7.017, 34.301, -90]
  MoveL 1298 to (-392.82, -100.42, 908) mm, rotated rx 180 ry 0 rz -90 deg; joints [54.576, -65.342, -124.737, 10.078, 35.424, -90]
  MoveL 1299 to (-390.65, -85.71, 903) mm, rotated rx 180 ry 0 rz -90 deg; joints [53.822, -66.818, -126.114, 12.933, 36.178, -90]
  MoveL 1300 to (-389.79, -71.39, 901) mm, rotated rx 180 ry 0 rz -90 deg; joints [53.531, -67.81, -127.707, 15.517, 36.469, -90]
  MoveL 1301 to (-384.6, -56.5, 889) mm, rotated rx 180 ry 0 rz -90 deg; joints [51.9, -70.932, -128.11, 19.042, 38.1, -90]
  MoveL 1302 to (-383.3, -42.41, 886) mm, rotated rx 180 ry 0 rz -90 deg; joints [51.52, -72.364, -129.393, 21.757, 38.48, -90]
  MoveL 1303 to (-380.27, -28.29, 879) mm, rotated rx 180 ry 0 rz -90 deg; joints [50.673, -74.689, -130.089, 24.778, 39.327, -90]
  MoveL 1304 to (-379.84, -14.49, 878) mm, rotated rx 180 ry 0 rz -90 deg; joints [50.556, -75.96, -131.45, 27.411, 39.444, -90]
  MoveL 1305 to (-376.38, -0.72, 870) mm, rotated rx 180 ry 0 rz -90 deg; joints [49.658, -78.661, -131.782, 30.443, 40.342, -90]
  MoveL 1306 to (-369.89, 12.7, 855) mm, rotated rx 180 ry 0 rz -90 deg; joints [48.129, -82.63, -130.948, 33.578, 41.871, -90]
  MoveL 1307 to (-369.89, 26.11, 855) mm, rotated rx 180 ry 0 rz -90 deg; joints [48.129, -84.011, -132.165, 36.176, 41.871, -90]
  MoveL 1308 to (-367.29, 39.24, 849) mm, rotated rx 180 ry 0 rz -90 deg; joints [47.567, -86.483, -132.39, 38.873, 42.433, -90]
  MoveL 1309 to (-363.83, 52.06, 841) mm, rotated rx 180 ry 0 rz -90 deg; joints [46.857, -89.288, -132.181, 41.469, 43.143, -90]
  MoveL 1310 to (-356.91, 64, 825) mm, rotated rx 180 ry 0 rz -90 deg; joints [45.558, -93.193, -130.522, 43.714, 44.442, -90]
  MoveL 1311 to (-359.07, 77.41, 830) mm, rotated rx 180 ry 0 rz -90 deg; joints [45.948, -94.163, -132.226, 46.389, 44.052, -90]
  MoveL 1312 to (-359.07, 90.42, 830) mm, rotated rx 180 ry 0 rz -90 deg; joints [45.948, -95.927, -133.036, 48.962, 44.052, -90]
  MoveL 1313 to (-353.02, 101.69, 816) mm, rotated rx 180 ry 0 rz -90 deg; joints [44.889, -99.39, -131.349, 50.739, 45.111, -90]
  MoveL 1314 to (-357.34, 115.89, 826) mm, rotated rx 180 ry 0 rz -90 deg; joints [45.635, -100.157, -133.744, 53.901, 44.365, -90]
  MoveL 1315 to (-370.66, -488.66, 889) mm, rotated rx 180 ry 0 rz -90 deg; joints [53.943, -85.49, -48.545, -45.966, 36.057, -90]
  MoveL 1316 to (-370.66, -474.72, 889) mm, rotated rx 180 ry 0 rz -90 deg; joints [53.943, -83.783, -52.87, -43.347, 36.057, -90]
  MoveL 1317 to (-368.57, -458.19, 884) mm, rotated rx 180 ry 0 rz -90 deg; joints [53.283, -82.691, -57.014, -40.295, 36.717, -90]
  MoveL 1318 to (-370.24, -446.33, 888) mm, rotated rx 180 ry 0 rz -90 deg; joints [53.808, -80.933, -60.66, -38.407, 36.192, -90]
  MoveL 1319 to (-367.74, -429.49, 882) mm, rotated rx 180 ry 0 rz -90 deg; joints [53.027, -80.252, -64.268, -35.48, 36.973, -90]
  MoveL 1320 to (-365.65, -413.3, 877) mm, rotated rx 180 ry 0 rz -90 deg; joints [52.406, -79.629, -67.604, -32.768, 37.594, -90]
  MoveL 1321 to (-368.99, -403.19, 885) mm, rotated rx 180 ry 0 rz -90 deg; joints [53.413, -77.705, -70.787, -31.508, 36.587, -90]
  MoveL 1322 to (-368.99, -389.31, 885) mm, rotated rx 180 ry 0 rz -90 deg; joints [53.413, -76.71, -73.856, -29.434, 36.587, -90]
  MoveL 1323 to (-371.07, -377.56, 890) mm, rotated rx 180 ry 0 rz -90 deg; joints [54.078, -75.202, -76.869, -27.929, 35.922, -90]
  MoveL 1324 to (-372.74, -365.24, 894) mm, rotated rx 180 ry 0 rz -90 deg; joints [54.632, -73.847, -79.806, -26.347, 35.368, -90]
  MoveL 1325 to (-374.41, -352.79, 898) mm, rotated rx 180 ry 0 rz -90 deg; joints [55.206, -72.529, -82.681, -24.79, 34.794, -90]
  MoveL 1326 to (-376.08, -340.21, 902) mm, rotated rx 180 ry 0 rz -90 deg; joints [55.801, -71.245, -85.502, -23.254, 34.199, -90]
  MoveL 1327 to (-376.49, -326.43, 903) mm, rotated rx 180 ry 0 rz -90 deg; joints [55.954, -70.388, -88.204, -21.408, 34.046, -90]
  MoveL 1328 to (-385.67, -319.88, 925) mm, rotated rx 180 ry 0 rz -90 deg; joints [59.714, -66.723, -91.337, -21.94, 30.286, -90]
  MoveL 1329 to (-379, -300.09, 909) mm, rotated rx 180 ry 0 rz -90 deg; joints [56.899, -68.272, -93.548, -18.18, 33.101, -90]
  MoveL 1330 to (-386.08, -291.18, 926) mm, rotated rx 180 ry 0 rz -90 deg; joints [59.906, -65.237, -96.587, -18.176, 30.094, -90]
  MoveL 1331 to (-384, -275.17, 921) mm, rotated rx 180 ry 0 rz -90 deg; joints [58.966, -65.401, -98.945, -15.655, 31.034, -90]
  MoveL 1332 to (-382.33, -259.59, 917) mm, rotated rx 180 ry 0 rz -90 deg; joints [58.249, -65.514, -101.232, -13.253, 31.751, -90]
  MoveL 1333 to (-396.51, -254.31, 951) mm, rotated rx 180 ry 0 rz -90 deg; joints [65.484, -59.65, -104.876, -15.474, 24.516, -90]
  MoveL 1334 to (-392.34, -236.88, 941) mm, rotated rx 180 ry 0 rz -90 deg; joints [63.055, -60.797, -106.986, -12.218, 26.945, -90]
  MoveL 1335 to (-389.42, -220.47, 934) mm, rotated rx 180 ry 0 rz -90 deg; joints [61.519, -61.581, -109.057, -9.361, 28.481, -90]
  MoveL 1336 to (-391.5, -206.92, 939) mm, rotated rx 180 ry 0 rz -90 deg; joints [62.603, -60.4, -111.612, -7.989, 27.397, -90]
  MoveL 1337 to (-386.5, -189.74, 927) mm, rotated rx 180 ry 0 rz -90 deg; joints [60.1, -62.289, -113.233, -4.478, 29.9, -90]
  MoveL 1338 to (-389.84, -176.72, 935) mm, rotated rx 180 ry 0 rz -90 deg; joints [61.731, -60.691, -115.909, -3.4, 28.269, -90]
  MoveL 1339 to (-387.75, -161.19, 930) mm, rotated rx 180 ry 0 rz -90 deg; joints [60.695, -61.545, -117.771, -0.684, 29.305, -90]
  MoveL 1340 to (-390.67, -147.71, 937) mm, rotated rx 180 ry 0 rz -90 deg; joints [62.162, -60.2, -120.375, 0.576, 27.838, -90]
  MoveL 1341 to (-387.75, -132.02, 930) mm, rotated rx 180 ry 0 rz -90 deg; joints [60.695, -61.662, -121.976, 3.637, 29.305, -90]
  MoveL 1342 to (-384.83, -116.55, 923) mm, rotated rx 180 ry 0 rz -90 deg; joints [59.336, -63.259, -123.449, 6.709, 30.664, -90]
  MoveL 1343 to (-382.33, -101.42, 917) mm, rotated rx 180 ry 0 rz -90 deg; joints [58.249, -64.791, -124.885, 9.676, 31.751, -90]
  MoveL 1344 to (-380.25, -86.56, 912) mm, rotated rx 180 ry 0 rz -90 deg; joints [57.393, -66.251, -126.303, 12.554, 32.607, -90]
  MoveL 1345 to (-374.83, -71.23, 899) mm, rotated rx 180 ry 0 rz -90 deg; joints [55.352, -69.425, -126.779, 16.204, 34.648, -90]
  MoveL 1346 to (-371.49, -56.62, 891) mm, rotated rx 180 ry 0 rz -90 deg; joints [54.215, -71.711, -127.597, 19.308, 35.785, -90]
  MoveL 1347 to (-368.16, -42.27, 883) mm, rotated rx 180 ry 0 rz -90 deg; joints [53.155, -74.092, -128.27, 22.362, 36.845, -90]
  MoveL 1348 to (-367.74, -28.39, 882) mm, rotated rx 180 ry 0 rz -90 deg; joints [53.027, -75.244, -129.69, 24.935, 36.973, -90]
  MoveL 1349 to (-371.49, -14.71, 891) mm, rotated rx 180 ry 0 rz -90 deg; joints [54.215, -74.608, -132.349, 26.957, 35.785, -90]
  MoveL 1350 to (-366.49, -0.73, 879) mm, rotated rx 180 ry 0 rz -90 deg; joints [52.652, -78.091, -132.206, 30.297, 37.348, -90]
  MoveL 1351 to (-357.73, 12.75, 858) mm, rotated rx 180 ry 0 rz -90 deg; joints [50.265, -83.105, -130.557, 33.662, 39.735, -90]
  MoveL 1352 to (-358.15, 26.23, 859) mm, rotated rx 180 ry 0 rz -90 deg; joints [50.37, -84.32, -131.92, 36.24, 39.63, -90]
  MoveL 1353 to (-355.65, 39.42, 853) mm, rotated rx 180 ry 0 rz -90 deg; joints [49.753, -86.78, -132.153, 38.932, 40.247, -90]
  MoveL 1354 to (-351.48, 52.18, 843) mm, rotated rx 180 ry 0 rz -90 deg; joints [48.783, -89.866, -131.634, 41.5, 41.217, -90]
  MoveL 1355 to (-351.89, 65.48, 844) mm, rotated rx 180 ry 0 rz -90 deg; joints [48.877, -91.357, -132.766, 44.123, 41.123, -90]
  MoveL 1356 to (-349.81, 78.25, 839) mm, rotated rx 180 ry 0 rz -90 deg; joints [48.415, -93.769, -132.841, 46.61, 41.585, -90]
  MoveL 1357 to (-346.06, 90.42, 830) mm, rotated rx 180 ry 0 rz -90 deg; joints [47.624, -96.685, -132.14, 48.825, 42.376, -90]
  MoveL 1358 to (-345.22, 103.19, 828) mm, rotated rx 180 ry 0 rz -90 deg; joints [47.455, -98.737, -132.526, 51.263, 42.545, -90]
  MoveL 1359 to (-344.39, 115.89, 826) mm, rotated rx 180 ry 0 rz -90 deg; joints [47.288, -100.84, -132.832, 53.672, 42.712, -90]
  MoveL 1360 to (-359.12, -477.92, 895) mm, rotated rx 180 ry 0 rz -90 deg; joints [56.69, -84.263, -51.818, -43.918, 33.31, -90]
  MoveL 1361 to (-358.32, -462.85, 893) mm, rotated rx 180 ry 0 rz -90 deg; joints [56.399, -82.849, -55.986, -41.165, 33.601, -90]
  MoveL 1362 to (-357.92, -448.35, 892) mm, rotated rx 180 ry 0 rz -90 deg; joints [56.255, -81.51, -59.83, -38.661, 33.745, -90]
  MoveL 1363 to (-359.12, -435.82, 895) mm, rotated rx 180 ry 0 rz -90 deg; joints [56.69, -79.913, -63.385, -36.702, 33.31, -90]
  MoveL 1364 to (-359.12, -421.78, 895) mm, rotated rx 180 ry 0 rz -90 deg; joints [56.69, -78.699, -66.819, -34.482, 33.31, -90]
  MoveL 1365 to (-358.72, -407.29, 894) mm, rotated rx 180 ry 0 rz -90 deg; joints [56.544, -77.685, -70.097, -32.218, 33.456, -90]
  MoveL 1366 to (-362.33, -397.23, 903) mm, rotated rx 180 ry 0 rz -90 deg; joints [57.906, -75.666, -73.249, -31.085, 32.094, -90]
  MoveL 1367 to (-361.13, -381.8, 900) mm, rotated rx 180 ry 0 rz -90 deg; joints [57.44, -75.016, -76.292, -28.691, 32.56, -90]
  MoveL 1368 to (-362.73, -369.32, 904) mm, rotated rx 180 ry 0 rz -90 deg; joints [58.064, -73.641, -79.274, -27.085, 31.936, -90]
  MoveL 1369 to (-367.15, -359.47, 915) mm, rotated rx 180 ry 0 rz -90 deg; joints [59.9, -71.457, -82.275, -26.269, 30.1, -90]
  MoveL 1370 to (-361.53, -339.84, 901) mm, rotated rx 180 ry 0 rz -90 deg; joints [57.594, -72.382, -84.841, -22.776, 32.406, -90]
  MoveL 1371 to (-365.14, -328.96, 910) mm, rotated rx 180 ry 0 rz -90 deg; joints [59.042, -70.506, -87.735, -21.759, 30.958, -90]
  MoveL 1372 to (-369.15, -318.15, 920) mm, rotated rx 180 ry 0 rz -90 deg; joints [60.799, -68.49, -90.624, -20.885, 29.201, -90]
  MoveL 1373 to (-371.56, -305.7, 926) mm, rotated rx 180 ry 0 rz -90 deg; joints [61.936, -67.004, -93.398, -19.598, 28.064, -90]
  MoveL 1374 to (-371.56, -291.18, 926) mm, rotated rx 180 ry 0 rz -90 deg; joints [61.936, -66.377, -95.979, -17.644, 28.064, -90]
  MoveL 1375 to (-373.57, -278.16, 931) mm, rotated rx 180 ry 0 rz -90 deg; joints [62.936, -65.081, -98.66, -16.259, 27.064, -90]
  MoveL 1376 to (-371.56, -262.14, 926) mm, rotated rx 180 ry 0 rz -90 deg; joints [61.936, -65.307, -100.961, -13.732, 28.064, -90]
  MoveL 1377 to (-378.38, -252.17, 943) mm, rotated rx 180 ry 0 rz -90 deg; joints [65.559, -62.224, -104.024, -13.752, 24.441, -90]
  MoveL 1378 to (-378.38, -237.38, 943) mm, rotated rx 180 ry 0 rz -90 deg; joints [65.559, -61.768, -106.456, -11.776, 24.441, -90]
  MoveL 1379 to (-389.22, -228.96, 970) mm, rotated rx 180 ry 0 rz -90 deg; joints [72.945, -56.825, -109.858, -13.317, 17.055, -90]
  MoveL 1380 to (-372.36, -117.18, 928) mm, rotated rx 180 ry 0 rz -90 deg; joints [62.33, -63.689, -123.136, 6.825, 27.67, -90]
  MoveL 1381 to (-367.95, -101.42, 917) mm, rotated rx 180 ry 0 rz -90 deg; joints [60.254, -66.168, -124.136, 10.304, 29.746, -90]
  MoveL 1382 to (-367.15, -86.85, 915) mm, rotated rx 180 ry 0 rz -90 deg; joints [59.9, -67.03, -125.824, 12.854, 30.1, -90]
  MoveL 1383 to (-363.54, -71.78, 906) mm, rotated rx 180 ry 0 rz -90 deg; joints [58.384, -69.377, -126.724, 16.1, 31.616, -90]
  MoveL 1384 to (-362.73, -57.45, 904) mm, rotated rx 180 ry 0 rz -90 deg; joints [58.064, -70.486, -128.24, 18.726, 31.936, -90]
  MoveL 1385 to (-361.53, -43.13, 901) mm, rotated rx 180 ry 0 rz -90 deg; joints [57.594, -71.909, -129.572, 21.482, 32.406, -90]
  MoveL 1386 to (-358.72, -28.78, 894) mm, rotated rx 180 ry 0 rz -90 deg; joints [56.544, -74.217, -130.333, 24.55, 33.456, -90]
  MoveL 1387 to (-360.33, -14.82, 898) mm, rotated rx 180 ry 0 rz -90 deg; joints [57.136, -74.552, -132.368, 26.92, 32.864, -90]
  MoveL 1388 to (-352.7, -0.73, 879) mm, rotated rx 180 ry 0 rz -90 deg; joints [54.491, -79.274, -131.315, 30.589, 35.509, -90]
  MoveL 1389 to (-348.29, 12.89, 868) mm, rotated rx 180 ry 0 rz -90 deg; joints [53.135, -82.489, -131.098, 33.588, 36.865, -90]
  MoveL 1390 to (-348.29, 26.51, 868) mm, rotated rx 180 ry 0 rz -90 deg; joints [53.135, -83.896, -132.335, 36.232, 36.865, -90]
  MoveL 1391 to (-345.48, 39.79, 861) mm, rotated rx 180 ry 0 rz -90 deg; joints [52.33, -86.534, -132.447, 38.982, 37.67, -90]
  MoveL 1392 to (-342.27, 52.8, 853) mm, rotated rx 180 ry 0 rz -90 deg; joints [51.46, -89.338, -132.277, 41.615, 38.54, -90]
  MoveL 1393 to (-342.67, 66.25, 854) mm, rotated rx 180 ry 0 rz -90 deg; joints [51.566, -90.871, -133.424, 44.295, 38.434, -90]
  MoveL 1394 to (-339.06, 78.81, 845) mm, rotated rx 180 ry 0 rz -90 deg; joints [50.638, -93.85, -132.87, 46.721, 39.362, -90]
  MoveL 1395 to (-334.65, 90.86, 834) mm, rotated rx 180 ry 0 rz -90 deg; joints [49.58, -97.006, -131.853, 48.859, 40.42, -90]
  MoveL 1396 to (-335.05, 104.06, 835) mm, rotated rx 180 ry 0 rz -90 deg; joints [49.673, -98.722, -132.749, 51.471, 40.327, -90]
  MoveL 1397 to (-341.62, -445.33, 886) mm, rotated rx 180 ry 0 rz -90 deg; joints [57.152, -83.088, -59.104, -37.809, 32.848, -90]
  MoveL 1398 to (-345.09, -435.82, 895) mm, rotated rx 180 ry 0 rz -90 deg; joints [58.454, -80.945, -62.584, -36.471, 31.546, -90]
  MoveL 1399 to (-348.94, -426.5, 905) mm, rotated rx 180 ry 0 rz -90 deg; joints [60.015, -78.745, -65.946, -35.31, 29.985, -90]
  MoveL 1400 to (-347.4, -410.48, 901) mm, rotated rx 180 ry 0 rz -90 deg; joints [59.376, -77.991, -69.321, -32.687, 30.625, -90]
  MoveL 1401 to (-349.33, -398.55, 906) mm, rotated rx 180 ry 0 rz -90 deg; joints [60.179, -76.401, -72.514, -31.086, 29.821, -90]
  MoveL 1402 to (-347.79, -382.65, 902) mm, rotated rx 180 ry 0 rz -90 deg; joints [59.534, -75.847, -75.578, -28.575, 30.466, -90]
  MoveL 1403 to (-355.88, -377.08, 923) mm, rotated rx 180 ry 0 rz -90 deg; joints [63.18, -72.551, -78.693, -28.756, 26.82, -90]
  MoveL 1404 to (-355.5, -362.22, 922) mm, rotated rx 180 ry 0 rz -90 deg; joints [62.99, -71.746, -81.647, -26.607, 27.01, -90]
  MoveL 1405 to (-357.04, -334.75, 926) mm, rotated rx 180 ry 0 rz -90 deg; joints [63.758, -69.615, -87.357, -23.028, 26.242, -90]
  MoveL 1406 to (-360.13, -322.99, 934) mm, rotated rx 180 ry 0 rz -90 deg; joints [65.379, -67.849, -90.229, -21.922, 24.621, -90]
  MoveL 1407 to (-357.43, -306.03, 927) mm, rotated rx 180 ry 0 rz -90 deg; joints [63.954, -68.076, -92.745, -19.179, 26.046, -90]
  MoveL 1408 to (-341.62, -0.73, 886) mm, rotated rx 180 ry 0 rz -90 deg; joints [57.152, -79.301, -131.294, 30.594, 32.848, -90]
  MoveL 1409 to (-338.53, 13.04, 878) mm, rotated rx 180 ry 0 rz -90 deg; joints [56.069, -81.992, -131.534, 33.527, 33.931, -90]
  MoveL 1410 to (-339.69, 26.9, 881) mm, rotated rx 180 ry 0 rz -90 deg; joints [56.467, -82.93, -133.225, 36.155, 33.533, -90]
  MoveL 1411 to (-336.99, 40.4, 874) mm, rotated rx 180 ry 0 rz -90 deg; joints [55.551, -85.614, -133.393, 39.007, 34.449, -90]
  MoveL 1412 to (-333.91, 53.61, 866) mm, rotated rx 180 ry 0 rz -90 deg; joints [54.56, -88.471, -133.277, 41.748, 35.44, -90]
  MoveL 1413 to (-333.91, 67.19, 866) mm, rotated rx 180 ry 0 rz -90 deg; joints [54.56, -90.204, -134.29, 44.495, 35.44, -90]
  MoveL 1414 to (-326.2, 78.9, 846) mm, rotated rx 180 ry 0 rz -90 deg; joints [52.314, -94.647, -132.001, 46.647, 37.686, -90]
  MoveL 1415 to (-323.11, 91.3, 838) mm, rotated rx 180 ry 0 rz -90 deg; joints [51.497, -97.388, -131.489, 48.877, 38.503, -90]
  MoveL 1416 to (-321.95, 104.06, 835) mm, rotated rx 180 ry 0 rz -90 deg; joints [51.202, -99.539, -131.707, 51.246, 38.798, -90]
  Set speed (1000.0 mm/s)
  MoveL 1417 to (-321.95, 104.06, 835) mm, rotated rx 180 ry 0 rz -90 deg; joints [51.202, -99.539, -131.707, 51.246, 38.798, -90]
  MoveL 1418 to (-321.95, 104.06, 935) mm, rotated rx 180 ry 0 rz -90 deg; joints [69.485, -89.01, -143.613, 52.623, 20.515, -90]
